// TIA Portal V20 export
DATA_BLOCK "HmiInterface"   // DB88
{ DB_Accessible_From_OPC_UA := 'FALSE' }
AUTHOR : ERsystem_FA2_DH. Kim
// stored: Access Published, DBAccessibleFromOPCUA false, DBAccessibleFromWebserver false, MemoryReserve 100, Namespace Unit1.Em7
   VAR
      em : "LAF_typeEmInterface";
      cm : Struct
         softCam : "Unit1.type_emRelations_em7_SoftCam";
         brakeTest : Struct
            sepaClampnCutterAxisZ : "LER_typeBrakeTestEmInterface";
            sepaGripperAxisZ : "LER_typeBrakeTestEmInterface";
            jrPusherAxisZ : "LER_typeBrakeTestEmInterface";
         END_STRUCT;
      END_STRUCT;
      sepaClamp : Struct
         jobs { S7_SetPoint := 'True'} : "LAF_typeJobsInterface";
         sequence { S7_SetPoint := 'True'} : "LAF_typeSequenceInterface";
      END_STRUCT;
      sepaGripper : Struct
         jobs { S7_SetPoint := 'True'} : "LAF_typeJobsInterface";
         sequence { S7_SetPoint := 'True'} : "LAF_typeSequenceInterface";
      END_STRUCT;
      jellyRollWinder : Struct
         jobs { S7_SetPoint := 'True'} : "LAF_typeJobsInterface";
         sequence { S7_SetPoint := 'True'} : "LAF_typeSequenceInterface";
      END_STRUCT;
      distance : Struct
         SepaClampToSepaGripperDisance : "LER_typeDistanceInterface";
         SepaGripperToSepaClampDisance : "LER_typeDistanceInterface";
         SepaGripperAxisCHomeDeg { S7_SetPoint := 'True'} : "LER_typeDistanceInterface";
         SepaGripperAxisXHomeDis { S7_SetPoint := 'True'} : "LER_typeDistanceInterface";
      END_STRUCT;
      cmSepaClampDetectSensor { S7_SetPoint := 'True'} : "LBC_typeDigitalSignalInterface";
      cmSepaGripperDetectSensor { S7_SetPoint := 'True'} : "LBC_typeDigitalSignalInterface";
      cmJRWinderDetectSensor { S7_SetPoint := 'True'} : "LBC_typeDigitalSignalInterface";
      cmSepaClampSafetyPinDetectSensor { S7_SetPoint := 'True'} : "LBC_typeDigitalSignalInterface";
      cmSepaGripperSafetyPinDetectSensor { S7_SetPoint := 'True'} : "LBC_typeDigitalSignalInterface";
   END_VAR
   VAR RETAIN
      cmSepaClampnCutterAxisX : "LBC_typeAxis64PosInterface";
      cmSepaClampnCutterAxisZ { S7_SetPoint := 'True'} : "LBC_typeAxis64PosInterface";
      cmSepaGripperAxisX : "LBC_typeAxis64PosInterface";
      cmSepaGripperAxisZ { S7_SetPoint := 'True'} : "LBC_typeAxis64PosInterface";
      cmSepaGripperAxisC : "LBC_typeAxis64PosInterface";
      cmJRWinderRearAxisY : "LBC_typeAxis64PosInterface";
      cmJRWinderFrontAxisY : "LBC_typeAxis64PosInterface";
      cmJRWinderAxisB { S7_SetPoint := 'True'} : "LBC_typeAxis64PosInterface";
      cmJRPusherAxisZ { S7_SetPoint := 'True'} : "LBC_typeAxis64PosInterface";
   END_VAR
   VAR
      cmSepaCutterUpDown { S7_SetPoint := 'True'} : "LBC_typeTwoWayActuatorInterface";
      cmSepaClampTopUpDown { S7_SetPoint := 'True'} : "LBC_typeTwoWayActuatorInterface";
      cmSepaClampBottomUpDown { S7_SetPoint := 'True'} : "LBC_typeTwoWayActuatorInterface";
      cmStackGripperOpenClose { S7_SetPoint := 'True'} : "LBC_typeTwoWayActuatorInterface";
      cmStackGripperFwdBwd { S7_SetPoint := 'True'} : "LBC_typeTwoWayActuatorInterface";
      cmJRWinderClampTopRearUpDown : "LBC_typeTwoWayActuatorInterface";
      cmJRWinderClampBtmRearUpDown : "LBC_typeTwoWayActuatorInterface";
      cmJRWinderClampTopFrontUpDown : "LBC_typeTwoWayActuatorInterface";
      cmJRWinderClampBtmFrontUpDown : "LBC_typeTwoWayActuatorInterface";
      cmPusherRollerUpDown : "LBC_typeTwoWayActuatorInterface";
      cmPusherRollerFwdBwd : "LBC_typeTwoWayActuatorInterface";
      cmHotWireCutter : "LER_typeHotWireCutterInterface";
      intCondition : Struct
         Axis_34 { S7_SetPoint := 'True'} : "LER.typeAxisIntlockAll";   // SepaClampnCutterAxisX
         Axis_35 { S7_SetPoint := 'True'} : "LER.typeAxisIntlockAll";   // SepaClampnCutterAxisZ
         Axis_36 { S7_SetPoint := 'True'} : "LER.typeAxisIntlockAll";   // SepaGripperAxisX
         Axis_37 { S7_SetPoint := 'True'} : "LER.typeAxisIntlockAll";   // SepaGripperAxisZ
         Axis_38 { S7_SetPoint := 'True'} : "LER.typeAxisIntlockAll";   // SepaGripperAxisC
         Axis_39 { S7_SetPoint := 'True'} : "LER.typeAxisIntlockAll";   // JRWinderFrontAxisY
         Axis_40 { S7_SetPoint := 'True'} : "LER.typeAxisIntlockAll";   // JRWinderRearAxisY
         Axis_41 { S7_SetPoint := 'True'} : "LER.typeAxisIntlockAll";   // JRWinderAxisB
         Axis_42 { S7_SetPoint := 'True'} : "LER.typeAxisIntlockAll";   // JRPusherAxisZ
         Axis_04 { S7_SetPoint := 'True'} : "LER.typeAxisIntlockAll";   // SepaClampnCutterAxisX
         Actuator_38 { S7_SetPoint := 'True'} : "LER.typeAxisActuatorCondition";   // SP
         Actuator_39 { S7_SetPoint := 'True'} : "LER.typeAxisActuatorCondition";   // SP
         Actuator_40 { S7_SetPoint := 'True'} : "LER.typeAxisActuatorCondition";   // JRWinderClampRightBtmUpDown
         Actuator_41 { S7_SetPoint := 'True'} : "LER.typeAxisActuatorCondition";   // JRWinderClampLeftBtmUpDown
         Actuator_42 { S7_SetPoint := 'True'} : "LER.typeAxisActuatorCondition";   // JRWinderClampLeftTopUpDown
         Actuator_43 { S7_SetPoint := 'True'} : "LER.typeAxisActuatorCondition";   // StackGripperFwdBwd
         Actuator_44 { S7_SetPoint := 'True'} : "LER.typeAxisActuatorCondition";   // SepaClampBottomUpDown
         Actuator_45 { S7_SetPoint := 'True'} : "LER.typeAxisActuatorCondition";   // SepaClampTopUpDown
         Actuator_46 { S7_SetPoint := 'True'} : "LER.typeAxisActuatorCondition";   // SepaCutterLeftUpDown
         Actuator_47 { S7_SetPoint := 'True'} : "LER.typeAxisActuatorCondition";   // JRWinderClampRightTopUpDown
         Actuator_48 { S7_SetPoint := 'True'} : "LER.typeAxisActuatorCondition";   // StackGripperOpenClose
         Actuator_49 { S7_SetPoint := 'True'} : "LER.typeAxisActuatorCondition";   // PusherRollerFwdBwd
      END_STRUCT;
   END_VAR
BEGIN
   em.interlinkMode.link := FALSE;
   em.interlinkMode.unlink := FALSE;
   em.interlinkMode.isLinked := TRUE;
   em.commands.enable := FALSE;
   em.commands.acknowledge := FALSE;
   em.commands.disableAlarms := FALSE;
   em.commands.activateSimulation := FALSE;
   em.commands.home := FALSE;
   em.commands.moveToInitialPosition := FALSE;
   em.commands.directModeControl := 16#0000_0001;
   em.commands.directStateControl := 16#0000_0004;
   em.status.enabled := TRUE;
   em.status.acknowledgeActive := FALSE;
   em.status.alarmsDisabled := FALSE;
   em.status.simulationActive := TRUE;
   em.status.safetyReleased := TRUE;
   em.status.initialized := FALSE;
   em.status.homed := FALSE;
   em.status.safeState := FALSE;
   em.status.stateComplete := FALSE;
   em.alarms.error := FALSE;
   em.alarms.warning := FALSE;
   em.alarms.info := FALSE;
   em.alarms.home := FALSE;
   cm.softCam.sepaClampnCutterAxisX.waitPos.inPos := TRUE;
   cm.softCam.sepaClampnCutterAxisX.waitPos.isBefore := FALSE;
   cm.softCam.sepaClampnCutterAxisX.waitPos.isAfter := FALSE;
   cm.softCam.sepaClampnCutterAxisX.sepaClampnCutPos.inPos := FALSE;
   cm.softCam.sepaClampnCutterAxisX.sepaClampnCutPos.isBefore := FALSE;
   cm.softCam.sepaClampnCutterAxisX.sepaClampnCutPos.isAfter := TRUE;
   cm.softCam.sepaClampnCutterAxisX.winderReadyPos.inPos := FALSE;
   cm.softCam.sepaClampnCutterAxisX.winderReadyPos.isBefore := TRUE;
   cm.softCam.sepaClampnCutterAxisX.winderReadyPos.isAfter := FALSE;
   cm.softCam.sepaClampnCutterAxisX.angle90.inPos := FALSE;
   cm.softCam.sepaClampnCutterAxisX.angle90.isBefore := TRUE;
   cm.softCam.sepaClampnCutterAxisX.angle90.isAfter := FALSE;
   cm.softCam.sepaClampnCutterAxisX.angle180.inPos := FALSE;
   cm.softCam.sepaClampnCutterAxisX.angle180.isBefore := TRUE;
   cm.softCam.sepaClampnCutterAxisX.angle180.isAfter := FALSE;
   cm.softCam.sepaClampnCutterAxisX.angle270.inPos := FALSE;
   cm.softCam.sepaClampnCutterAxisX.angle270.isBefore := TRUE;
   cm.softCam.sepaClampnCutterAxisX.angle270.isAfter := FALSE;
   cm.softCam.sepaClampnCutterAxisX.angle360.inPos := FALSE;
   cm.softCam.sepaClampnCutterAxisX.angle360.isBefore := TRUE;
   cm.softCam.sepaClampnCutterAxisX.angle360.isAfter := FALSE;
   cm.softCam.sepaClampnCutterAxisX.Pos8.inPos := FALSE;
   cm.softCam.sepaClampnCutterAxisX.Pos8.isBefore := FALSE;
   cm.softCam.sepaClampnCutterAxisX.Pos8.isAfter := TRUE;
   cm.softCam.sepaClampnCutterAxisX.Pos9.inPos := FALSE;
   cm.softCam.sepaClampnCutterAxisX.Pos9.isBefore := FALSE;
   cm.softCam.sepaClampnCutterAxisX.Pos9.isAfter := TRUE;
   cm.softCam.sepaClampnCutterAxisX.Pos10.inPos := FALSE;
   cm.softCam.sepaClampnCutterAxisX.Pos10.isBefore := FALSE;
   cm.softCam.sepaClampnCutterAxisX.Pos10.isAfter := TRUE;
   cm.softCam.sepaClampnCutterAxisX.Pos11.inPos := FALSE;
   cm.softCam.sepaClampnCutterAxisX.Pos11.isBefore := FALSE;
   cm.softCam.sepaClampnCutterAxisX.Pos11.isAfter := TRUE;
   cm.softCam.sepaClampnCutterAxisX.Pos12.inPos := FALSE;
   cm.softCam.sepaClampnCutterAxisX.Pos12.isBefore := FALSE;
   cm.softCam.sepaClampnCutterAxisX.Pos12.isAfter := TRUE;
   cm.softCam.sepaClampnCutterAxisX.Pos13.inPos := FALSE;
   cm.softCam.sepaClampnCutterAxisX.Pos13.isBefore := FALSE;
   cm.softCam.sepaClampnCutterAxisX.Pos13.isAfter := TRUE;
   cm.softCam.sepaClampnCutterAxisX.Pos14.inPos := FALSE;
   cm.softCam.sepaClampnCutterAxisX.Pos14.isBefore := FALSE;
   cm.softCam.sepaClampnCutterAxisX.Pos14.isAfter := TRUE;
   cm.softCam.sepaClampnCutterAxisX.Pos15.inPos := FALSE;
   cm.softCam.sepaClampnCutterAxisX.Pos15.isBefore := FALSE;
   cm.softCam.sepaClampnCutterAxisX.Pos15.isAfter := TRUE;
   cm.softCam.sepaClampnCutterAxisZ.waitPos.inPos := TRUE;
   cm.softCam.sepaClampnCutterAxisZ.waitPos.isBefore := FALSE;
   cm.softCam.sepaClampnCutterAxisZ.waitPos.isAfter := FALSE;
   cm.softCam.sepaClampnCutterAxisZ.sepaCutnClampPos.inPos := FALSE;
   cm.softCam.sepaClampnCutterAxisZ.sepaCutnClampPos.isBefore := TRUE;
   cm.softCam.sepaClampnCutterAxisZ.sepaCutnClampPos.isAfter := FALSE;
   cm.softCam.sepaClampnCutterAxisZ.winderReadyPos.inPos := FALSE;
   cm.softCam.sepaClampnCutterAxisZ.winderReadyPos.isBefore := TRUE;
   cm.softCam.sepaClampnCutterAxisZ.winderReadyPos.isAfter := FALSE;
   cm.softCam.sepaClampnCutterAxisZ.verticalPos.inPos := FALSE;
   cm.softCam.sepaClampnCutterAxisZ.verticalPos.isBefore := FALSE;
   cm.softCam.sepaClampnCutterAxisZ.verticalPos.isAfter := TRUE;
   cm.softCam.sepaClampnCutterAxisZ.horizonPos.inPos := TRUE;
   cm.softCam.sepaClampnCutterAxisZ.horizonPos.isBefore := FALSE;
   cm.softCam.sepaClampnCutterAxisZ.horizonPos.isAfter := FALSE;
   cm.softCam.sepaClampnCutterAxisZ.Pos5.inPos := TRUE;
   cm.softCam.sepaClampnCutterAxisZ.Pos5.isBefore := FALSE;
   cm.softCam.sepaClampnCutterAxisZ.Pos5.isAfter := FALSE;
   cm.softCam.sepaClampnCutterAxisZ.Pos6.inPos := TRUE;
   cm.softCam.sepaClampnCutterAxisZ.Pos6.isBefore := FALSE;
   cm.softCam.sepaClampnCutterAxisZ.Pos6.isAfter := FALSE;
   cm.softCam.sepaClampnCutterAxisZ.Pos7.inPos := TRUE;
   cm.softCam.sepaClampnCutterAxisZ.Pos7.isBefore := FALSE;
   cm.softCam.sepaClampnCutterAxisZ.Pos7.isAfter := FALSE;
   cm.softCam.sepaClampnCutterAxisZ.Pos8.inPos := TRUE;
   cm.softCam.sepaClampnCutterAxisZ.Pos8.isBefore := FALSE;
   cm.softCam.sepaClampnCutterAxisZ.Pos8.isAfter := FALSE;
   cm.softCam.sepaClampnCutterAxisZ.Pos9.inPos := TRUE;
   cm.softCam.sepaClampnCutterAxisZ.Pos9.isBefore := FALSE;
   cm.softCam.sepaClampnCutterAxisZ.Pos9.isAfter := FALSE;
   cm.softCam.sepaClampnCutterAxisZ.Pos10.inPos := TRUE;
   cm.softCam.sepaClampnCutterAxisZ.Pos10.isBefore := FALSE;
   cm.softCam.sepaClampnCutterAxisZ.Pos10.isAfter := FALSE;
   cm.softCam.sepaClampnCutterAxisZ.Pos11.inPos := TRUE;
   cm.softCam.sepaClampnCutterAxisZ.Pos11.isBefore := FALSE;
   cm.softCam.sepaClampnCutterAxisZ.Pos11.isAfter := FALSE;
   cm.softCam.sepaClampnCutterAxisZ.Pos12.inPos := TRUE;
   cm.softCam.sepaClampnCutterAxisZ.Pos12.isBefore := FALSE;
   cm.softCam.sepaClampnCutterAxisZ.Pos12.isAfter := FALSE;
   cm.softCam.sepaClampnCutterAxisZ.Pos13.inPos := TRUE;
   cm.softCam.sepaClampnCutterAxisZ.Pos13.isBefore := FALSE;
   cm.softCam.sepaClampnCutterAxisZ.Pos13.isAfter := FALSE;
   cm.softCam.sepaClampnCutterAxisZ.Pos14.inPos := TRUE;
   cm.softCam.sepaClampnCutterAxisZ.Pos14.isBefore := FALSE;
   cm.softCam.sepaClampnCutterAxisZ.Pos14.isAfter := FALSE;
   cm.softCam.sepaClampnCutterAxisZ.Pos15.inPos := TRUE;
   cm.softCam.sepaClampnCutterAxisZ.Pos15.isBefore := FALSE;
   cm.softCam.sepaClampnCutterAxisZ.Pos15.isAfter := FALSE;
   cm.softCam.sepaGripperAxisX.waitPos.inPos := TRUE;
   cm.softCam.sepaGripperAxisX.waitPos.isBefore := FALSE;
   cm.softCam.sepaGripperAxisX.waitPos.isAfter := FALSE;
   cm.softCam.sepaGripperAxisX.pickUpPOs.inPos := FALSE;
   cm.softCam.sepaGripperAxisX.pickUpPOs.isBefore := TRUE;
   cm.softCam.sepaGripperAxisX.pickUpPOs.isAfter := FALSE;
   cm.softCam.sepaGripperAxisX.sepaTailPos.inPos := FALSE;
   cm.softCam.sepaGripperAxisX.sepaTailPos.isBefore := TRUE;
   cm.softCam.sepaGripperAxisX.sepaTailPos.isAfter := FALSE;
   cm.softCam.sepaGripperAxisX.jrWinderPos.inPos := FALSE;
   cm.softCam.sepaGripperAxisX.jrWinderPos.isBefore := TRUE;
   cm.softCam.sepaGripperAxisX.jrWinderPos.isAfter := FALSE;
   cm.softCam.sepaGripperAxisX.turn_ngDischargePos.inPos := FALSE;
   cm.softCam.sepaGripperAxisX.turn_ngDischargePos.isBefore := TRUE;
   cm.softCam.sepaGripperAxisX.turn_ngDischargePos.isAfter := FALSE;
   cm.softCam.sepaGripperAxisX.avoidPos.inPos := TRUE;
   cm.softCam.sepaGripperAxisX.avoidPos.isBefore := FALSE;
   cm.softCam.sepaGripperAxisX.avoidPos.isAfter := FALSE;
   cm.softCam.sepaGripperAxisX.okDisChargePos.inPos := FALSE;
   cm.softCam.sepaGripperAxisX.okDisChargePos.isBefore := FALSE;
   cm.softCam.sepaGripperAxisX.okDisChargePos.isAfter := TRUE;
   cm.softCam.sepaGripperAxisX.ngSepaTailPos.inPos := FALSE;
   cm.softCam.sepaGripperAxisX.ngSepaTailPos.isBefore := FALSE;
   cm.softCam.sepaGripperAxisX.ngSepaTailPos.isAfter := TRUE;
   cm.softCam.sepaGripperAxisX.jrWinderZonePos.inPos := FALSE;
   cm.softCam.sepaGripperAxisX.jrWinderZonePos.isBefore := FALSE;
   cm.softCam.sepaGripperAxisX.jrWinderZonePos.isAfter := TRUE;
   cm.softCam.sepaGripperAxisX.gripperAxisCCollisionZonePos.inPos := FALSE;
   cm.softCam.sepaGripperAxisX.gripperAxisCCollisionZonePos.isBefore := FALSE;
   cm.softCam.sepaGripperAxisX.gripperAxisCCollisionZonePos.isAfter := TRUE;
   cm.softCam.sepaGripperAxisX.anodePnPZonePos.inPos := FALSE;
   cm.softCam.sepaGripperAxisX.anodePnPZonePos.isBefore := FALSE;
   cm.softCam.sepaGripperAxisX.anodePnPZonePos.isAfter := TRUE;
   cm.softCam.sepaGripperAxisX.pickUpBeforePos.inPos := FALSE;
   cm.softCam.sepaGripperAxisX.pickUpBeforePos.isBefore := FALSE;
   cm.softCam.sepaGripperAxisX.pickUpBeforePos.isAfter := TRUE;
   cm.softCam.sepaGripperAxisX.Pos12.inPos := FALSE;
   cm.softCam.sepaGripperAxisX.Pos12.isBefore := FALSE;
   cm.softCam.sepaGripperAxisX.Pos12.isAfter := TRUE;
   cm.softCam.sepaGripperAxisX.Pos13.inPos := FALSE;
   cm.softCam.sepaGripperAxisX.Pos13.isBefore := FALSE;
   cm.softCam.sepaGripperAxisX.Pos13.isAfter := TRUE;
   cm.softCam.sepaGripperAxisX.Pos14.inPos := FALSE;
   cm.softCam.sepaGripperAxisX.Pos14.isBefore := FALSE;
   cm.softCam.sepaGripperAxisX.Pos14.isAfter := TRUE;
   cm.softCam.sepaGripperAxisX.Pos15.inPos := FALSE;
   cm.softCam.sepaGripperAxisX.Pos15.isBefore := FALSE;
   cm.softCam.sepaGripperAxisX.Pos15.isAfter := TRUE;
   cm.softCam.sepaGripperAxisZ.waitPos.inPos := TRUE;
   cm.softCam.sepaGripperAxisZ.waitPos.isBefore := FALSE;
   cm.softCam.sepaGripperAxisZ.waitPos.isAfter := FALSE;
   cm.softCam.sepaGripperAxisZ.jrWinderPos.inPos := FALSE;
   cm.softCam.sepaGripperAxisZ.jrWinderPos.isBefore := TRUE;
   cm.softCam.sepaGripperAxisZ.jrWinderPos.isAfter := FALSE;
   cm.softCam.sepaGripperAxisZ.turnPos.inPos := FALSE;
   cm.softCam.sepaGripperAxisZ.turnPos.isBefore := TRUE;
   cm.softCam.sepaGripperAxisZ.turnPos.isAfter := FALSE;
   cm.softCam.sepaGripperAxisZ.jrWinderRePickUpPos.inPos := FALSE;
   cm.softCam.sepaGripperAxisZ.jrWinderRePickUpPos.isBefore := TRUE;
   cm.softCam.sepaGripperAxisZ.jrWinderRePickUpPos.isAfter := FALSE;
   cm.softCam.sepaGripperAxisZ.okDisChargePos.inPos := FALSE;
   cm.softCam.sepaGripperAxisZ.okDisChargePos.isBefore := TRUE;
   cm.softCam.sepaGripperAxisZ.okDisChargePos.isAfter := FALSE;
   cm.softCam.sepaGripperAxisZ.ngDischargePos.inPos := FALSE;
   cm.softCam.sepaGripperAxisZ.ngDischargePos.isBefore := TRUE;
   cm.softCam.sepaGripperAxisZ.ngDischargePos.isAfter := FALSE;
   cm.softCam.sepaGripperAxisZ.pickUpPos.inPos := FALSE;
   cm.softCam.sepaGripperAxisZ.pickUpPos.isBefore := TRUE;
   cm.softCam.sepaGripperAxisZ.pickUpPos.isAfter := FALSE;
   cm.softCam.sepaGripperAxisZ.Pos7.inPos := TRUE;
   cm.softCam.sepaGripperAxisZ.Pos7.isBefore := FALSE;
   cm.softCam.sepaGripperAxisZ.Pos7.isAfter := FALSE;
   cm.softCam.sepaGripperAxisZ.Pos8.inPos := TRUE;
   cm.softCam.sepaGripperAxisZ.Pos8.isBefore := FALSE;
   cm.softCam.sepaGripperAxisZ.Pos8.isAfter := FALSE;
   cm.softCam.sepaGripperAxisZ.Pos9.inPos := TRUE;
   cm.softCam.sepaGripperAxisZ.Pos9.isBefore := FALSE;
   cm.softCam.sepaGripperAxisZ.Pos9.isAfter := FALSE;
   cm.softCam.sepaGripperAxisZ.Pos10.inPos := TRUE;
   cm.softCam.sepaGripperAxisZ.Pos10.isBefore := FALSE;
   cm.softCam.sepaGripperAxisZ.Pos10.isAfter := FALSE;
   cm.softCam.sepaGripperAxisZ.Pos11.inPos := TRUE;
   cm.softCam.sepaGripperAxisZ.Pos11.isBefore := FALSE;
   cm.softCam.sepaGripperAxisZ.Pos11.isAfter := FALSE;
   cm.softCam.sepaGripperAxisZ.Pos12.inPos := TRUE;
   cm.softCam.sepaGripperAxisZ.Pos12.isBefore := FALSE;
   cm.softCam.sepaGripperAxisZ.Pos12.isAfter := FALSE;
   cm.softCam.sepaGripperAxisZ.Pos13.inPos := TRUE;
   cm.softCam.sepaGripperAxisZ.Pos13.isBefore := FALSE;
   cm.softCam.sepaGripperAxisZ.Pos13.isAfter := FALSE;
   cm.softCam.sepaGripperAxisZ.Pos14.inPos := TRUE;
   cm.softCam.sepaGripperAxisZ.Pos14.isBefore := FALSE;
   cm.softCam.sepaGripperAxisZ.Pos14.isAfter := FALSE;
   cm.softCam.sepaGripperAxisZ.Pos15.inPos := TRUE;
   cm.softCam.sepaGripperAxisZ.Pos15.isBefore := FALSE;
   cm.softCam.sepaGripperAxisZ.Pos15.isAfter := FALSE;
   cm.softCam.sepaGripperAxisC.waitPos.inPos := TRUE;
   cm.softCam.sepaGripperAxisC.waitPos.isBefore := FALSE;
   cm.softCam.sepaGripperAxisC.waitPos.isAfter := FALSE;
   cm.softCam.sepaGripperAxisC.okDischargePos.inPos := FALSE;
   cm.softCam.sepaGripperAxisC.okDischargePos.isBefore := TRUE;
   cm.softCam.sepaGripperAxisC.okDischargePos.isAfter := FALSE;
   cm.softCam.sepaGripperAxisC.ngDischargePos.inPos := FALSE;
   cm.softCam.sepaGripperAxisC.ngDischargePos.isBefore := TRUE;
   cm.softCam.sepaGripperAxisC.ngDischargePos.isAfter := FALSE;
   cm.softCam.sepaGripperAxisC.Pos3.inPos := TRUE;
   cm.softCam.sepaGripperAxisC.Pos3.isBefore := FALSE;
   cm.softCam.sepaGripperAxisC.Pos3.isAfter := FALSE;
   cm.softCam.sepaGripperAxisC.Pos4.inPos := TRUE;
   cm.softCam.sepaGripperAxisC.Pos4.isBefore := FALSE;
   cm.softCam.sepaGripperAxisC.Pos4.isAfter := FALSE;
   cm.softCam.sepaGripperAxisC.Pos5.inPos := TRUE;
   cm.softCam.sepaGripperAxisC.Pos5.isBefore := FALSE;
   cm.softCam.sepaGripperAxisC.Pos5.isAfter := FALSE;
   cm.softCam.sepaGripperAxisC.Pos6.inPos := TRUE;
   cm.softCam.sepaGripperAxisC.Pos6.isBefore := FALSE;
   cm.softCam.sepaGripperAxisC.Pos6.isAfter := FALSE;
   cm.softCam.sepaGripperAxisC.Pos7.inPos := TRUE;
   cm.softCam.sepaGripperAxisC.Pos7.isBefore := FALSE;
   cm.softCam.sepaGripperAxisC.Pos7.isAfter := FALSE;
   cm.softCam.sepaGripperAxisC.Pos8.inPos := TRUE;
   cm.softCam.sepaGripperAxisC.Pos8.isBefore := FALSE;
   cm.softCam.sepaGripperAxisC.Pos8.isAfter := FALSE;
   cm.softCam.sepaGripperAxisC.Pos9.inPos := TRUE;
   cm.softCam.sepaGripperAxisC.Pos9.isBefore := FALSE;
   cm.softCam.sepaGripperAxisC.Pos9.isAfter := FALSE;
   cm.softCam.sepaGripperAxisC.Pos10.inPos := TRUE;
   cm.softCam.sepaGripperAxisC.Pos10.isBefore := FALSE;
   cm.softCam.sepaGripperAxisC.Pos10.isAfter := FALSE;
   cm.softCam.sepaGripperAxisC.Pos11.inPos := TRUE;
   cm.softCam.sepaGripperAxisC.Pos11.isBefore := FALSE;
   cm.softCam.sepaGripperAxisC.Pos11.isAfter := FALSE;
   cm.softCam.sepaGripperAxisC.Pos12.inPos := TRUE;
   cm.softCam.sepaGripperAxisC.Pos12.isBefore := FALSE;
   cm.softCam.sepaGripperAxisC.Pos12.isAfter := FALSE;
   cm.softCam.sepaGripperAxisC.Pos13.inPos := TRUE;
   cm.softCam.sepaGripperAxisC.Pos13.isBefore := FALSE;
   cm.softCam.sepaGripperAxisC.Pos13.isAfter := FALSE;
   cm.softCam.sepaGripperAxisC.Pos14.inPos := TRUE;
   cm.softCam.sepaGripperAxisC.Pos14.isBefore := FALSE;
   cm.softCam.sepaGripperAxisC.Pos14.isAfter := FALSE;
   cm.softCam.sepaGripperAxisC.Pos15.inPos := TRUE;
   cm.softCam.sepaGripperAxisC.Pos15.isBefore := FALSE;
   cm.softCam.sepaGripperAxisC.Pos15.isAfter := FALSE;
   cm.softCam.jrWinderRearAxisY.waitPos.inPos := TRUE;
   cm.softCam.jrWinderRearAxisY.waitPos.isBefore := FALSE;
   cm.softCam.jrWinderRearAxisY.waitPos.isAfter := FALSE;
   cm.softCam.jrWinderRearAxisY.clampPos.inPos := FALSE;
   cm.softCam.jrWinderRearAxisY.clampPos.isBefore := TRUE;
   cm.softCam.jrWinderRearAxisY.clampPos.isAfter := FALSE;
   cm.softCam.jrWinderRearAxisY.Pos2.inPos := TRUE;
   cm.softCam.jrWinderRearAxisY.Pos2.isBefore := FALSE;
   cm.softCam.jrWinderRearAxisY.Pos2.isAfter := FALSE;
   cm.softCam.jrWinderRearAxisY.Pos3.inPos := TRUE;
   cm.softCam.jrWinderRearAxisY.Pos3.isBefore := FALSE;
   cm.softCam.jrWinderRearAxisY.Pos3.isAfter := FALSE;
   cm.softCam.jrWinderRearAxisY.Pos4.inPos := TRUE;
   cm.softCam.jrWinderRearAxisY.Pos4.isBefore := FALSE;
   cm.softCam.jrWinderRearAxisY.Pos4.isAfter := FALSE;
   cm.softCam.jrWinderRearAxisY.Pos5.inPos := TRUE;
   cm.softCam.jrWinderRearAxisY.Pos5.isBefore := FALSE;
   cm.softCam.jrWinderRearAxisY.Pos5.isAfter := FALSE;
   cm.softCam.jrWinderRearAxisY.Pos6.inPos := TRUE;
   cm.softCam.jrWinderRearAxisY.Pos6.isBefore := FALSE;
   cm.softCam.jrWinderRearAxisY.Pos6.isAfter := FALSE;
   cm.softCam.jrWinderRearAxisY.Pos7.inPos := TRUE;
   cm.softCam.jrWinderRearAxisY.Pos7.isBefore := FALSE;
   cm.softCam.jrWinderRearAxisY.Pos7.isAfter := FALSE;
   cm.softCam.jrWinderRearAxisY.Pos8.inPos := TRUE;
   cm.softCam.jrWinderRearAxisY.Pos8.isBefore := FALSE;
   cm.softCam.jrWinderRearAxisY.Pos8.isAfter := FALSE;
   cm.softCam.jrWinderRearAxisY.Pos9.inPos := TRUE;
   cm.softCam.jrWinderRearAxisY.Pos9.isBefore := FALSE;
   cm.softCam.jrWinderRearAxisY.Pos9.isAfter := FALSE;
   cm.softCam.jrWinderRearAxisY.Pos10.inPos := TRUE;
   cm.softCam.jrWinderRearAxisY.Pos10.isBefore := FALSE;
   cm.softCam.jrWinderRearAxisY.Pos10.isAfter := FALSE;
   cm.softCam.jrWinderRearAxisY.Pos11.inPos := TRUE;
   cm.softCam.jrWinderRearAxisY.Pos11.isBefore := FALSE;
   cm.softCam.jrWinderRearAxisY.Pos11.isAfter := FALSE;
   cm.softCam.jrWinderRearAxisY.Pos12.inPos := TRUE;
   cm.softCam.jrWinderRearAxisY.Pos12.isBefore := FALSE;
   cm.softCam.jrWinderRearAxisY.Pos12.isAfter := FALSE;
   cm.softCam.jrWinderRearAxisY.Pos13.inPos := TRUE;
   cm.softCam.jrWinderRearAxisY.Pos13.isBefore := FALSE;
   cm.softCam.jrWinderRearAxisY.Pos13.isAfter := FALSE;
   cm.softCam.jrWinderRearAxisY.Pos14.inPos := TRUE;
   cm.softCam.jrWinderRearAxisY.Pos14.isBefore := FALSE;
   cm.softCam.jrWinderRearAxisY.Pos14.isAfter := FALSE;
   cm.softCam.jrWinderRearAxisY.Pos15.inPos := TRUE;
   cm.softCam.jrWinderRearAxisY.Pos15.isBefore := FALSE;
   cm.softCam.jrWinderRearAxisY.Pos15.isAfter := FALSE;
   cm.softCam.jrWinderFrontAxisY.waitPos.inPos := TRUE;
   cm.softCam.jrWinderFrontAxisY.waitPos.isBefore := FALSE;
   cm.softCam.jrWinderFrontAxisY.waitPos.isAfter := FALSE;
   cm.softCam.jrWinderFrontAxisY.clampPos.inPos := FALSE;
   cm.softCam.jrWinderFrontAxisY.clampPos.isBefore := TRUE;
   cm.softCam.jrWinderFrontAxisY.clampPos.isAfter := FALSE;
   cm.softCam.jrWinderFrontAxisY.Pos2.inPos := TRUE;
   cm.softCam.jrWinderFrontAxisY.Pos2.isBefore := FALSE;
   cm.softCam.jrWinderFrontAxisY.Pos2.isAfter := FALSE;
   cm.softCam.jrWinderFrontAxisY.Pos3.inPos := TRUE;
   cm.softCam.jrWinderFrontAxisY.Pos3.isBefore := FALSE;
   cm.softCam.jrWinderFrontAxisY.Pos3.isAfter := FALSE;
   cm.softCam.jrWinderFrontAxisY.Pos4.inPos := TRUE;
   cm.softCam.jrWinderFrontAxisY.Pos4.isBefore := FALSE;
   cm.softCam.jrWinderFrontAxisY.Pos4.isAfter := FALSE;
   cm.softCam.jrWinderFrontAxisY.Pos5.inPos := TRUE;
   cm.softCam.jrWinderFrontAxisY.Pos5.isBefore := FALSE;
   cm.softCam.jrWinderFrontAxisY.Pos5.isAfter := FALSE;
   cm.softCam.jrWinderFrontAxisY.Pos6.inPos := TRUE;
   cm.softCam.jrWinderFrontAxisY.Pos6.isBefore := FALSE;
   cm.softCam.jrWinderFrontAxisY.Pos6.isAfter := FALSE;
   cm.softCam.jrWinderFrontAxisY.Pos7.inPos := TRUE;
   cm.softCam.jrWinderFrontAxisY.Pos7.isBefore := FALSE;
   cm.softCam.jrWinderFrontAxisY.Pos7.isAfter := FALSE;
   cm.softCam.jrWinderFrontAxisY.Pos8.inPos := TRUE;
   cm.softCam.jrWinderFrontAxisY.Pos8.isBefore := FALSE;
   cm.softCam.jrWinderFrontAxisY.Pos8.isAfter := FALSE;
   cm.softCam.jrWinderFrontAxisY.Pos9.inPos := TRUE;
   cm.softCam.jrWinderFrontAxisY.Pos9.isBefore := FALSE;
   cm.softCam.jrWinderFrontAxisY.Pos9.isAfter := FALSE;
   cm.softCam.jrWinderFrontAxisY.Pos10.inPos := TRUE;
   cm.softCam.jrWinderFrontAxisY.Pos10.isBefore := FALSE;
   cm.softCam.jrWinderFrontAxisY.Pos10.isAfter := FALSE;
   cm.softCam.jrWinderFrontAxisY.Pos11.inPos := TRUE;
   cm.softCam.jrWinderFrontAxisY.Pos11.isBefore := FALSE;
   cm.softCam.jrWinderFrontAxisY.Pos11.isAfter := FALSE;
   cm.softCam.jrWinderFrontAxisY.Pos12.inPos := TRUE;
   cm.softCam.jrWinderFrontAxisY.Pos12.isBefore := FALSE;
   cm.softCam.jrWinderFrontAxisY.Pos12.isAfter := FALSE;
   cm.softCam.jrWinderFrontAxisY.Pos13.inPos := TRUE;
   cm.softCam.jrWinderFrontAxisY.Pos13.isBefore := FALSE;
   cm.softCam.jrWinderFrontAxisY.Pos13.isAfter := FALSE;
   cm.softCam.jrWinderFrontAxisY.Pos14.inPos := TRUE;
   cm.softCam.jrWinderFrontAxisY.Pos14.isBefore := FALSE;
   cm.softCam.jrWinderFrontAxisY.Pos14.isAfter := FALSE;
   cm.softCam.jrWinderFrontAxisY.Pos15.inPos := TRUE;
   cm.softCam.jrWinderFrontAxisY.Pos15.isBefore := FALSE;
   cm.softCam.jrWinderFrontAxisY.Pos15.isAfter := FALSE;
   cm.softCam.jrWinderAxisB.waitPos.inPos := TRUE;
   cm.softCam.jrWinderAxisB.waitPos.isBefore := FALSE;
   cm.softCam.jrWinderAxisB.waitPos.isAfter := FALSE;
   cm.softCam.jrWinderAxisB.angle90.inPos := FALSE;
   cm.softCam.jrWinderAxisB.angle90.isBefore := TRUE;
   cm.softCam.jrWinderAxisB.angle90.isAfter := FALSE;
   cm.softCam.jrWinderAxisB.angle180.inPos := FALSE;
   cm.softCam.jrWinderAxisB.angle180.isBefore := TRUE;
   cm.softCam.jrWinderAxisB.angle180.isAfter := FALSE;
   cm.softCam.jrWinderAxisB.angle270.inPos := FALSE;
   cm.softCam.jrWinderAxisB.angle270.isBefore := TRUE;
   cm.softCam.jrWinderAxisB.angle270.isAfter := FALSE;
   cm.softCam.jrWinderAxisB.angle360.inPos := TRUE;
   cm.softCam.jrWinderAxisB.angle360.isBefore := FALSE;
   cm.softCam.jrWinderAxisB.angle360.isAfter := FALSE;
   cm.softCam.jrWinderAxisB.angle450.inPos := TRUE;
   cm.softCam.jrWinderAxisB.angle450.isBefore := FALSE;
   cm.softCam.jrWinderAxisB.angle450.isAfter := FALSE;
   cm.softCam.jrWinderAxisB.angle540.inPos := TRUE;
   cm.softCam.jrWinderAxisB.angle540.isBefore := FALSE;
   cm.softCam.jrWinderAxisB.angle540.isAfter := FALSE;
   cm.softCam.jrWinderAxisB.Pos9.inPos := TRUE;
   cm.softCam.jrWinderAxisB.Pos9.isBefore := FALSE;
   cm.softCam.jrWinderAxisB.Pos9.isAfter := FALSE;
   cm.softCam.jrWinderAxisB.Pos10.inPos := TRUE;
   cm.softCam.jrWinderAxisB.Pos10.isBefore := FALSE;
   cm.softCam.jrWinderAxisB.Pos10.isAfter := FALSE;
   cm.softCam.jrWinderAxisB.Pos11.inPos := TRUE;
   cm.softCam.jrWinderAxisB.Pos11.isBefore := FALSE;
   cm.softCam.jrWinderAxisB.Pos11.isAfter := FALSE;
   cm.softCam.jrWinderAxisB.Pos12.inPos := TRUE;
   cm.softCam.jrWinderAxisB.Pos12.isBefore := FALSE;
   cm.softCam.jrWinderAxisB.Pos12.isAfter := FALSE;
   cm.softCam.jrWinderAxisB.Pos13.inPos := TRUE;
   cm.softCam.jrWinderAxisB.Pos13.isBefore := FALSE;
   cm.softCam.jrWinderAxisB.Pos13.isAfter := FALSE;
   cm.softCam.jrWinderAxisB.Pos14.inPos := TRUE;
   cm.softCam.jrWinderAxisB.Pos14.isBefore := FALSE;
   cm.softCam.jrWinderAxisB.Pos14.isAfter := FALSE;
   cm.softCam.jrWinderAxisB.Pos15.inPos := TRUE;
   cm.softCam.jrWinderAxisB.Pos15.isBefore := FALSE;
   cm.softCam.jrWinderAxisB.Pos15.isAfter := FALSE;
   cm.softCam.jrPusherAxisZ.waitPos.inPos := TRUE;
   cm.softCam.jrPusherAxisZ.waitPos.isBefore := FALSE;
   cm.softCam.jrPusherAxisZ.waitPos.isAfter := FALSE;
   cm.softCam.jrPusherAxisZ.downPos.inPos := FALSE;
   cm.softCam.jrPusherAxisZ.downPos.isBefore := TRUE;
   cm.softCam.jrPusherAxisZ.downPos.isAfter := FALSE;
   cm.softCam.jrPusherAxisZ.verticalPos.inPos := FALSE;
   cm.softCam.jrPusherAxisZ.verticalPos.isBefore := FALSE;
   cm.softCam.jrPusherAxisZ.verticalPos.isAfter := TRUE;
   cm.softCam.jrPusherAxisZ.horizonPos.inPos := TRUE;
   cm.softCam.jrPusherAxisZ.horizonPos.isBefore := FALSE;
   cm.softCam.jrPusherAxisZ.horizonPos.isAfter := FALSE;
   cm.softCam.jrPusherAxisZ.Pos4.inPos := TRUE;
   cm.softCam.jrPusherAxisZ.Pos4.isBefore := FALSE;
   cm.softCam.jrPusherAxisZ.Pos4.isAfter := FALSE;
   cm.softCam.jrPusherAxisZ.Pos5.inPos := TRUE;
   cm.softCam.jrPusherAxisZ.Pos5.isBefore := FALSE;
   cm.softCam.jrPusherAxisZ.Pos5.isAfter := FALSE;
   cm.softCam.jrPusherAxisZ.Pos6.inPos := TRUE;
   cm.softCam.jrPusherAxisZ.Pos6.isBefore := FALSE;
   cm.softCam.jrPusherAxisZ.Pos6.isAfter := FALSE;
   cm.softCam.jrPusherAxisZ.Pos7.inPos := TRUE;
   cm.softCam.jrPusherAxisZ.Pos7.isBefore := FALSE;
   cm.softCam.jrPusherAxisZ.Pos7.isAfter := FALSE;
   cm.softCam.jrPusherAxisZ.Pos8.inPos := TRUE;
   cm.softCam.jrPusherAxisZ.Pos8.isBefore := FALSE;
   cm.softCam.jrPusherAxisZ.Pos8.isAfter := FALSE;
   cm.softCam.jrPusherAxisZ.Pos9.inPos := TRUE;
   cm.softCam.jrPusherAxisZ.Pos9.isBefore := FALSE;
   cm.softCam.jrPusherAxisZ.Pos9.isAfter := FALSE;
   cm.softCam.jrPusherAxisZ.Pos10.inPos := TRUE;
   cm.softCam.jrPusherAxisZ.Pos10.isBefore := FALSE;
   cm.softCam.jrPusherAxisZ.Pos10.isAfter := FALSE;
   cm.softCam.jrPusherAxisZ.Pos11.inPos := TRUE;
   cm.softCam.jrPusherAxisZ.Pos11.isBefore := FALSE;
   cm.softCam.jrPusherAxisZ.Pos11.isAfter := FALSE;
   cm.softCam.jrPusherAxisZ.Pos12.inPos := TRUE;
   cm.softCam.jrPusherAxisZ.Pos12.isBefore := FALSE;
   cm.softCam.jrPusherAxisZ.Pos12.isAfter := FALSE;
   cm.softCam.jrPusherAxisZ.Pos13.inPos := TRUE;
   cm.softCam.jrPusherAxisZ.Pos13.isBefore := FALSE;
   cm.softCam.jrPusherAxisZ.Pos13.isAfter := FALSE;
   cm.softCam.jrPusherAxisZ.Pos14.inPos := TRUE;
   cm.softCam.jrPusherAxisZ.Pos14.isBefore := FALSE;
   cm.softCam.jrPusherAxisZ.Pos14.isAfter := FALSE;
   cm.softCam.jrPusherAxisZ.Pos15.inPos := TRUE;
   cm.softCam.jrPusherAxisZ.Pos15.isBefore := FALSE;
   cm.softCam.jrPusherAxisZ.Pos15.isAfter := FALSE;
   cm.brakeTest.sepaClampnCutterAxisZ.commands.start := FALSE;
   cm.brakeTest.sepaClampnCutterAxisZ.commands.stop := FALSE;
   cm.brakeTest.sepaClampnCutterAxisZ.monitoring.error := FALSE;
   cm.brakeTest.sepaClampnCutterAxisZ.monitoring.ready := FALSE;
   cm.brakeTest.sepaClampnCutterAxisZ.monitoring.busy := FALSE;
   cm.brakeTest.sepaClampnCutterAxisZ.monitoring.complete := FALSE;
   cm.brakeTest.sepaClampnCutterAxisZ.monitoring.brakeSelected := FALSE;
   cm.brakeTest.sepaClampnCutterAxisZ.monitoring.brakeActive := FALSE;
   cm.brakeTest.sepaClampnCutterAxisZ.monitoring.brakeResult := FALSE;
   cm.brakeTest.sepaClampnCutterAxisZ.monitoring.brakeCompleted := FALSE;
   cm.brakeTest.sepaClampnCutterAxisZ.monitoring."step" := 0;
   cm.brakeTest.sepaGripperAxisZ.commands.start := FALSE;
   cm.brakeTest.sepaGripperAxisZ.commands.stop := FALSE;
   cm.brakeTest.sepaGripperAxisZ.monitoring.error := FALSE;
   cm.brakeTest.sepaGripperAxisZ.monitoring.ready := FALSE;
   cm.brakeTest.sepaGripperAxisZ.monitoring.busy := FALSE;
   cm.brakeTest.sepaGripperAxisZ.monitoring.complete := FALSE;
   cm.brakeTest.sepaGripperAxisZ.monitoring.brakeSelected := FALSE;
   cm.brakeTest.sepaGripperAxisZ.monitoring.brakeActive := FALSE;
   cm.brakeTest.sepaGripperAxisZ.monitoring.brakeResult := FALSE;
   cm.brakeTest.sepaGripperAxisZ.monitoring.brakeCompleted := FALSE;
   cm.brakeTest.sepaGripperAxisZ.monitoring."step" := 0;
   cm.brakeTest.jrPusherAxisZ.commands.start := FALSE;
   cm.brakeTest.jrPusherAxisZ.commands.stop := FALSE;
   cm.brakeTest.jrPusherAxisZ.monitoring.error := FALSE;
   cm.brakeTest.jrPusherAxisZ.monitoring.ready := FALSE;
   cm.brakeTest.jrPusherAxisZ.monitoring.busy := FALSE;
   cm.brakeTest.jrPusherAxisZ.monitoring.complete := FALSE;
   cm.brakeTest.jrPusherAxisZ.monitoring.brakeSelected := FALSE;
   cm.brakeTest.jrPusherAxisZ.monitoring.brakeActive := FALSE;
   cm.brakeTest.jrPusherAxisZ.monitoring.brakeResult := FALSE;
   cm.brakeTest.jrPusherAxisZ.monitoring.brakeCompleted := FALSE;
   cm.brakeTest.jrPusherAxisZ.monitoring."step" := 0;
   sepaClamp.jobs.commands.setJobNumber := 0;
   sepaClamp.jobs.commands.reset := FALSE;
   sepaClamp.jobs.status.activeJobNumber := 1;
   sepaClamp.jobs.status.previousCycleJobNumber := 1;
   sepaClamp.jobs.status.manualControlEnabled := FALSE;
   sepaClamp.jobs.status.memoryJobTime := 16#0000_4E90_6672_4E37;
   sepaClamp.sequence.commands.setAutomaticMode := FALSE;
   sepaClamp.sequence.commands.setSingleStepMode := FALSE;
   sepaClamp.sequence.commands.off := FALSE;
   sepaClamp.sequence.commands.initialize := FALSE;
   sepaClamp.sequence.commands.start := FALSE;
   sepaClamp.sequence.commands.immediateStop := FALSE;
   sepaClamp.sequence.commands.hold := FALSE;
   sepaClamp.sequence.commands.nextStep := FALSE;
   sepaClamp.sequence.commands.interlockStepChange := FALSE;
   sepaClamp.sequence.monitoring.automaticMode := TRUE;
   sepaClamp.sequence.monitoring.singleStepMode := FALSE;
   sepaClamp.sequence.monitoring.currentStep := 101;
   sepaClamp.sequence.monitoring.nextStep := 101;
   sepaClamp.sequence.monitoring.previousStep := 1;
   sepaClamp.sequence.monitoring.currentStepSTRING := 'N/A';
   sepaClamp.sequence.monitoring.nextStepSTRING := 'N/A';
   sepaClamp.sequence.monitoring.previousStepSTRING := 'N/A';
   sepaClamp.sequence.monitoring.inStepIdle := FALSE;
   sepaClamp.sequence.monitoring.inStepStopped := FALSE;
   sepaClamp.sequence.monitoring.seqActive := TRUE;
   sepaClamp.sequence.monitoring.stepActive := TRUE;
   sepaClamp.sequence.monitoring.stepComplete := FALSE;
   sepaClamp.sequence.monitoring.executionEnabled := FALSE;
   sepaClamp.sequence.monitoring.initRequired := FALSE;
   sepaClamp.sequence.monitoring.stepChangeReleased := TRUE;
   sepaClamp.sequence.monitoring.justSteppedPulse := FALSE;
   sepaClamp.sequence.monitoring.manualControlEnabled := FALSE;
   sepaClamp.sequence.monitoring.manualModeChangeEnabled := FALSE;
   sepaClamp.sequence.monitoring.memoryStepTimer := 16#0000_4E90_6828_A4A1;
   sepaGripper.jobs.commands.setJobNumber := 0;
   sepaGripper.jobs.commands.reset := FALSE;
   sepaGripper.jobs.status.activeJobNumber := 0;
   sepaGripper.jobs.status.previousCycleJobNumber := 0;
   sepaGripper.jobs.status.manualControlEnabled := FALSE;
   sepaGripper.jobs.status.memoryJobTime := 16#0000_4E92_AEA1_93D2;
   sepaGripper.sequence.commands.setAutomaticMode := FALSE;
   sepaGripper.sequence.commands.setSingleStepMode := FALSE;
   sepaGripper.sequence.commands.off := FALSE;
   sepaGripper.sequence.commands.initialize := FALSE;
   sepaGripper.sequence.commands.start := FALSE;
   sepaGripper.sequence.commands.immediateStop := FALSE;
   sepaGripper.sequence.commands.hold := FALSE;
   sepaGripper.sequence.commands.nextStep := FALSE;
   sepaGripper.sequence.commands.interlockStepChange := FALSE;
   sepaGripper.sequence.monitoring.automaticMode := TRUE;
   sepaGripper.sequence.monitoring.singleStepMode := FALSE;
   sepaGripper.sequence.monitoring.currentStep := 1;
   sepaGripper.sequence.monitoring.nextStep := 1;
   sepaGripper.sequence.monitoring.previousStep := 190;
   sepaGripper.sequence.monitoring.currentStepSTRING := 'N/A';
   sepaGripper.sequence.monitoring.nextStepSTRING := 'N/A';
   sepaGripper.sequence.monitoring.previousStepSTRING := 'N/A';
   sepaGripper.sequence.monitoring.inStepIdle := TRUE;
   sepaGripper.sequence.monitoring.inStepStopped := FALSE;
   sepaGripper.sequence.monitoring.seqActive := TRUE;
   sepaGripper.sequence.monitoring.stepActive := TRUE;
   sepaGripper.sequence.monitoring.stepComplete := FALSE;
   sepaGripper.sequence.monitoring.executionEnabled := TRUE;
   sepaGripper.sequence.monitoring.initRequired := FALSE;
   sepaGripper.sequence.monitoring.stepChangeReleased := TRUE;
   sepaGripper.sequence.monitoring.justSteppedPulse := FALSE;
   sepaGripper.sequence.monitoring.manualControlEnabled := FALSE;
   sepaGripper.sequence.monitoring.manualModeChangeEnabled := FALSE;
   sepaGripper.sequence.monitoring.memoryStepTimer := 16#0000_4E92_AEA0_D6D2;
   jellyRollWinder.jobs.commands.setJobNumber := 0;
   jellyRollWinder.jobs.commands.reset := FALSE;
   jellyRollWinder.jobs.status.activeJobNumber := 0;
   jellyRollWinder.jobs.status.previousCycleJobNumber := 0;
   jellyRollWinder.jobs.status.manualControlEnabled := FALSE;
   jellyRollWinder.jobs.status.memoryJobTime := 16#0000_4E90_62D8_99E4;
   jellyRollWinder.sequence.commands.setAutomaticMode := FALSE;
   jellyRollWinder.sequence.commands.setSingleStepMode := FALSE;
   jellyRollWinder.sequence.commands.off := FALSE;
   jellyRollWinder.sequence.commands.initialize := FALSE;
   jellyRollWinder.sequence.commands.start := FALSE;
   jellyRollWinder.sequence.commands.immediateStop := FALSE;
   jellyRollWinder.sequence.commands.hold := FALSE;
   jellyRollWinder.sequence.commands.nextStep := FALSE;
   jellyRollWinder.sequence.commands.interlockStepChange := FALSE;
   jellyRollWinder.sequence.monitoring.automaticMode := TRUE;
   jellyRollWinder.sequence.monitoring.singleStepMode := FALSE;
   jellyRollWinder.sequence.monitoring.currentStep := 1;
   jellyRollWinder.sequence.monitoring.nextStep := 1;
   jellyRollWinder.sequence.monitoring.previousStep := 190;
   jellyRollWinder.sequence.monitoring.currentStepSTRING := 'N/A';
   jellyRollWinder.sequence.monitoring.nextStepSTRING := 'N/A';
   jellyRollWinder.sequence.monitoring.previousStepSTRING := 'N/A';
   jellyRollWinder.sequence.monitoring.inStepIdle := TRUE;
   jellyRollWinder.sequence.monitoring.inStepStopped := FALSE;
   jellyRollWinder.sequence.monitoring.seqActive := TRUE;
   jellyRollWinder.sequence.monitoring.stepActive := TRUE;
   jellyRollWinder.sequence.monitoring.stepComplete := FALSE;
   jellyRollWinder.sequence.monitoring.executionEnabled := TRUE;
   jellyRollWinder.sequence.monitoring.initRequired := FALSE;
   jellyRollWinder.sequence.monitoring.stepChangeReleased := TRUE;
   jellyRollWinder.sequence.monitoring.justSteppedPulse := FALSE;
   jellyRollWinder.sequence.monitoring.manualControlEnabled := FALSE;
   jellyRollWinder.sequence.monitoring.manualModeChangeEnabled := FALSE;
   jellyRollWinder.sequence.monitoring.memoryStepTimer := 16#0000_4E90_62D7_E3E5;
   distance.SepaClampToSepaGripperDisance.setValue.direction := FALSE;
   distance.SepaClampToSepaGripperDisance.setValue.distanceLimitSV := 0.0;
   distance.SepaClampToSepaGripperDisance.setValue.distancePTPSV := 0.0;
   distance.SepaClampToSepaGripperDisance.processValue.distanceOutPos := FALSE;
   distance.SepaClampToSepaGripperDisance.processValue.distanceLimitPV := 0.0;
   distance.SepaClampToSepaGripperDisance.processValue.currentDistance := -200.0;
   distance.SepaGripperToSepaClampDisance.setValue.direction := FALSE;
   distance.SepaGripperToSepaClampDisance.setValue.distanceLimitSV := 0.0;
   distance.SepaGripperToSepaClampDisance.setValue.distancePTPSV := 0.0;
   distance.SepaGripperToSepaClampDisance.processValue.distanceOutPos := FALSE;
   distance.SepaGripperToSepaClampDisance.processValue.distanceLimitPV := 0.0;
   distance.SepaGripperToSepaClampDisance.processValue.currentDistance := -200.0;
   distance.SepaGripperAxisCHomeDeg.setValue.direction := FALSE;
   distance.SepaGripperAxisCHomeDeg.setValue.distanceLimitSV := 0.0;
   distance.SepaGripperAxisCHomeDeg.setValue.distancePTPSV := 0.0;
   distance.SepaGripperAxisCHomeDeg.processValue.distanceOutPos := FALSE;
   distance.SepaGripperAxisCHomeDeg.processValue.distanceLimitPV := 0.0;
   distance.SepaGripperAxisCHomeDeg.processValue.currentDistance := 0.0;
   distance.SepaGripperAxisXHomeDis.setValue.direction := FALSE;
   distance.SepaGripperAxisXHomeDis.setValue.distanceLimitSV := 0.0;
   distance.SepaGripperAxisXHomeDis.setValue.distancePTPSV := 0.0;
   distance.SepaGripperAxisXHomeDis.processValue.distanceOutPos := FALSE;
   distance.SepaGripperAxisXHomeDis.processValue.distanceLimitPV := 0.0;
   distance.SepaGripperAxisXHomeDis.processValue.currentDistance := 0.0;
   cmSepaClampDetectSensor.commands.refreshConfiguration := FALSE;
   cmSepaClampDetectSensor.commands.editConfiguration := FALSE;
   cmSepaClampDetectSensor.commands.saveConfiguration := FALSE;
   cmSepaClampDetectSensor.commands.reset := FALSE;
   cmSepaClampDetectSensor.monitoring.enable := TRUE;
   cmSepaClampDetectSensor.monitoring.referenceDesignator := WSTRING#'DigitalSignal';
   cmSepaClampDetectSensor.monitoring.simulation := FALSE;
   cmSepaClampDetectSensor.monitoring.processValue := FALSE;
   cmSepaClampDetectSensor.monitoring.error := FALSE;
   cmSepaClampDetectSensor.monitoring.status := 16#0000;
   cmSepaClampDetectSensor.configuration.referenceDesignator := WSTRING#'DigitalSignal';
   cmSepaClampDetectSensor.configuration.onDelay := T#0MS;
   cmSepaClampDetectSensor.configuration.offDelay := T#0MS;
   cmSepaClampDetectSensor.configuration.default := FALSE;
   cmSepaClampDetectSensor.configuration.invertProcessValue := FALSE;
   cmSepaClampDetectSensor.configuration.disableAlarms := FALSE;
   cmSepaGripperDetectSensor.commands.refreshConfiguration := FALSE;
   cmSepaGripperDetectSensor.commands.editConfiguration := FALSE;
   cmSepaGripperDetectSensor.commands.saveConfiguration := FALSE;
   cmSepaGripperDetectSensor.commands.reset := FALSE;
   cmSepaGripperDetectSensor.monitoring.enable := TRUE;
   cmSepaGripperDetectSensor.monitoring.referenceDesignator := WSTRING#'DigitalSignal';
   cmSepaGripperDetectSensor.monitoring.simulation := FALSE;
   cmSepaGripperDetectSensor.monitoring.processValue := FALSE;
   cmSepaGripperDetectSensor.monitoring.error := FALSE;
   cmSepaGripperDetectSensor.monitoring.status := 16#0000;
   cmSepaGripperDetectSensor.configuration.referenceDesignator := WSTRING#'DigitalSignal';
   cmSepaGripperDetectSensor.configuration.onDelay := T#0MS;
   cmSepaGripperDetectSensor.configuration.offDelay := T#0MS;
   cmSepaGripperDetectSensor.configuration.default := FALSE;
   cmSepaGripperDetectSensor.configuration.invertProcessValue := FALSE;
   cmSepaGripperDetectSensor.configuration.disableAlarms := FALSE;
   cmJRWinderDetectSensor.commands.refreshConfiguration := FALSE;
   cmJRWinderDetectSensor.commands.editConfiguration := FALSE;
   cmJRWinderDetectSensor.commands.saveConfiguration := FALSE;
   cmJRWinderDetectSensor.commands.reset := FALSE;
   cmJRWinderDetectSensor.monitoring.enable := TRUE;
   cmJRWinderDetectSensor.monitoring.referenceDesignator := WSTRING#'DigitalSignal';
   cmJRWinderDetectSensor.monitoring.simulation := FALSE;
   cmJRWinderDetectSensor.monitoring.processValue := FALSE;
   cmJRWinderDetectSensor.monitoring.error := FALSE;
   cmJRWinderDetectSensor.monitoring.status := 16#0000;
   cmJRWinderDetectSensor.configuration.referenceDesignator := WSTRING#'DigitalSignal';
   cmJRWinderDetectSensor.configuration.onDelay := T#0MS;
   cmJRWinderDetectSensor.configuration.offDelay := T#0MS;
   cmJRWinderDetectSensor.configuration.default := FALSE;
   cmJRWinderDetectSensor.configuration.invertProcessValue := FALSE;
   cmJRWinderDetectSensor.configuration.disableAlarms := FALSE;
   cmSepaClampSafetyPinDetectSensor.commands.refreshConfiguration := FALSE;
   cmSepaClampSafetyPinDetectSensor.commands.editConfiguration := FALSE;
   cmSepaClampSafetyPinDetectSensor.commands.saveConfiguration := FALSE;
   cmSepaClampSafetyPinDetectSensor.commands.reset := FALSE;
   cmSepaClampSafetyPinDetectSensor.monitoring.enable := TRUE;
   cmSepaClampSafetyPinDetectSensor.monitoring.referenceDesignator := WSTRING#'DigitalSignal';
   cmSepaClampSafetyPinDetectSensor.monitoring.simulation := FALSE;
   cmSepaClampSafetyPinDetectSensor.monitoring.processValue := FALSE;
   cmSepaClampSafetyPinDetectSensor.monitoring.error := FALSE;
   cmSepaClampSafetyPinDetectSensor.monitoring.status := 16#0000;
   cmSepaClampSafetyPinDetectSensor.configuration.referenceDesignator := WSTRING#'DigitalSignal';
   cmSepaClampSafetyPinDetectSensor.configuration.onDelay := T#0MS;
   cmSepaClampSafetyPinDetectSensor.configuration.offDelay := T#0MS;
   cmSepaClampSafetyPinDetectSensor.configuration.default := FALSE;
   cmSepaClampSafetyPinDetectSensor.configuration.invertProcessValue := FALSE;
   cmSepaClampSafetyPinDetectSensor.configuration.disableAlarms := FALSE;
   cmSepaGripperSafetyPinDetectSensor.commands.refreshConfiguration := FALSE;
   cmSepaGripperSafetyPinDetectSensor.commands.editConfiguration := FALSE;
   cmSepaGripperSafetyPinDetectSensor.commands.saveConfiguration := FALSE;
   cmSepaGripperSafetyPinDetectSensor.commands.reset := FALSE;
   cmSepaGripperSafetyPinDetectSensor.monitoring.enable := TRUE;
   cmSepaGripperSafetyPinDetectSensor.monitoring.referenceDesignator := WSTRING#'DigitalSignal';
   cmSepaGripperSafetyPinDetectSensor.monitoring.simulation := FALSE;
   cmSepaGripperSafetyPinDetectSensor.monitoring.processValue := FALSE;
   cmSepaGripperSafetyPinDetectSensor.monitoring.error := FALSE;
   cmSepaGripperSafetyPinDetectSensor.monitoring.status := 16#0000;
   cmSepaGripperSafetyPinDetectSensor.configuration.referenceDesignator := WSTRING#'DigitalSignal';
   cmSepaGripperSafetyPinDetectSensor.configuration.onDelay := T#0MS;
   cmSepaGripperSafetyPinDetectSensor.configuration.offDelay := T#0MS;
   cmSepaGripperSafetyPinDetectSensor.configuration.default := FALSE;
   cmSepaGripperSafetyPinDetectSensor.configuration.invertProcessValue := FALSE;
   cmSepaGripperSafetyPinDetectSensor.configuration.disableAlarms := FALSE;
   cmSepaClampnCutterAxisX.commandConfiguration.generalSettings.stopOnError := TRUE;
   cmSepaClampnCutterAxisX.commandConfiguration.generalSettings.resetWithRestart := FALSE;
   cmSepaClampnCutterAxisX.commandConfiguration.generalSettings.abortWaitingSyncCmd := TRUE;
   cmSepaClampnCutterAxisX.commandConfiguration.power.startMode := 1;
   cmSepaClampnCutterAxisX.commandConfiguration.power.stopMode := 0;
   cmSepaClampnCutterAxisX.commandConfiguration.power.syncMotionSimulation := FALSE;
   cmSepaClampnCutterAxisX.commandConfiguration.power.syncMotionSimulationExtendedMode := -1;
   cmSepaClampnCutterAxisX.commandConfiguration.jog.velocity := 0.0;
   cmSepaClampnCutterAxisX.commandConfiguration.jog.acceleration := -1.0;
   cmSepaClampnCutterAxisX.commandConfiguration.jog.deceleration := -1.0;
   cmSepaClampnCutterAxisX.commandConfiguration.jog.jerk := -1.0;
   cmSepaClampnCutterAxisX.commandConfiguration.jog.positionControlled := TRUE;
   cmSepaClampnCutterAxisX.commandConfiguration.jog.increment := 0.0;
   cmSepaClampnCutterAxisX.commandConfiguration.jog.mode := 0;
   cmSepaClampnCutterAxisX.commandConfiguration.moveVelocity.velocity := 0.0;
   cmSepaClampnCutterAxisX.commandConfiguration.moveVelocity.acceleration := -1.0;
   cmSepaClampnCutterAxisX.commandConfiguration.moveVelocity.deceleration := -1.0;
   cmSepaClampnCutterAxisX.commandConfiguration.moveVelocity.jerk := -1.0;
   cmSepaClampnCutterAxisX.commandConfiguration.moveVelocity.direction := 0;
   cmSepaClampnCutterAxisX.commandConfiguration.moveVelocity.positionControlled := TRUE;
   cmSepaClampnCutterAxisX.commandConfiguration.moveVelocity.velocityChangeOnTheFly := FALSE;
   cmSepaClampnCutterAxisX.commandConfiguration.stop.deceleration := -1.0;
   cmSepaClampnCutterAxisX.commandConfiguration.stop.jerk := -1.0;
   cmSepaClampnCutterAxisX.commandConfiguration.stop.abortAcceleration := FALSE;
   cmSepaClampnCutterAxisX.commandConfiguration.fastStop.deceleration := -1.0;
   cmSepaClampnCutterAxisX.commandConfiguration.fastStop.jerk := -1.0;
   cmSepaClampnCutterAxisX.commandConfiguration.fastStop.abortAcceleration := FALSE;
   cmSepaClampnCutterAxisX.commandConfiguration.fastStop.replaceStopPossible := FALSE;
   cmSepaClampnCutterAxisX.commandConfiguration.torqueLimiting.limit := -1.0;
   cmSepaClampnCutterAxisX.commandConfiguration.torqueLimiting.mode := 0;
   cmSepaClampnCutterAxisX.commandConfiguration.homing.position := 0.0;
   cmSepaClampnCutterAxisX.commandConfiguration.homing.mode := 0;
   cmSepaClampnCutterAxisX.commandConfiguration.homing.sensor := 0;
   cmSepaClampnCutterAxisX.commandConfiguration.homing.extendedMode := -1;
   cmSepaClampnCutterAxisX.commandConfiguration.homing.extendedModeTorqueLimit := 0.0;
   cmSepaClampnCutterAxisX.commandConfiguration.homing.extendedModeTargetPosition := 0.0;
   cmSepaClampnCutterAxisX.commandConfiguration.posRelative.distance := 0.0;
   cmSepaClampnCutterAxisX.commandConfiguration.posRelative.velocity := -1.0;
   cmSepaClampnCutterAxisX.commandConfiguration.posRelative.acceleration := -1.0;
   cmSepaClampnCutterAxisX.commandConfiguration.posRelative.deceleration := -1.0;
   cmSepaClampnCutterAxisX.commandConfiguration.posRelative.jerk := -1.0;
   cmSepaClampnCutterAxisX.commandConfiguration.posRelative.direction := 0;
   cmSepaClampnCutterAxisX.commandConfiguration.posAbsolute.position := 0.0;
   cmSepaClampnCutterAxisX.commandConfiguration.posAbsolute.velocity := -1.0;
   cmSepaClampnCutterAxisX.commandConfiguration.posAbsolute.acceleration := -1.0;
   cmSepaClampnCutterAxisX.commandConfiguration.posAbsolute.deceleration := -1.0;
   cmSepaClampnCutterAxisX.commandConfiguration.posAbsolute.jerk := -1.0;
   cmSepaClampnCutterAxisX.commandConfiguration.posAbsolute.direction := 1;
   cmSepaClampnCutterAxisX.commandConfiguration.posAbsolute.positionChangeOnTheFly := FALSE;
   cmSepaClampnCutterAxisX.commandConfiguration.posAbsolute.velocityChangeOnTheFly := FALSE;
   cmSepaClampnCutterAxisX.commandConfiguration.posSuperimposed.distance := 0.0;
   cmSepaClampnCutterAxisX.commandConfiguration.posSuperimposed.velocityDiff := -1.0;
   cmSepaClampnCutterAxisX.commandConfiguration.posSuperimposed.acceleration := -1.0;
   cmSepaClampnCutterAxisX.commandConfiguration.posSuperimposed.deceleration := -1.0;
   cmSepaClampnCutterAxisX.commandConfiguration.posSuperimposed.jerk := -1.0;
   cmSepaClampnCutterAxisX.commandConfiguration.posSuperimposed.direction := 0;
   cmSepaClampnCutterAxisX.commandConfiguration.haltSuperimposed.deceleration := -1.0;
   cmSepaClampnCutterAxisX.commandConfiguration.haltSuperimposed.jerk := -1.0;
   cmSepaClampnCutterAxisX.commandConfiguration.haltSuperimposed.abortAcceleration := FALSE;
   cmSepaClampnCutterAxisX.commandConfiguration.gearInRelative.ratioNumerator := 1;
   cmSepaClampnCutterAxisX.commandConfiguration.gearInRelative.ratioDenominator := 1;
   cmSepaClampnCutterAxisX.commandConfiguration.gearInRelative.acceleration := -1.0;
   cmSepaClampnCutterAxisX.commandConfiguration.gearInRelative.deceleration := -1.0;
   cmSepaClampnCutterAxisX.commandConfiguration.gearInRelative.jerk := -1.0;
   cmSepaClampnCutterAxisX.commandConfiguration.gearInRelative.ratioChangeOnTheFly := FALSE;
   cmSepaClampnCutterAxisX.commandConfiguration.gearInAbsolute.ratioNumerator := 1;
   cmSepaClampnCutterAxisX.commandConfiguration.gearInAbsolute.ratioDenominator := 1;
   cmSepaClampnCutterAxisX.commandConfiguration.gearInAbsolute.masterSyncPosition := 0.0;
   cmSepaClampnCutterAxisX.commandConfiguration.gearInAbsolute.slaveSyncPosition := 0.0;
   cmSepaClampnCutterAxisX.commandConfiguration.gearInAbsolute.syncProfileReference := 1;
   cmSepaClampnCutterAxisX.commandConfiguration.gearInAbsolute.masterStartDistance := 0.0;
   cmSepaClampnCutterAxisX.commandConfiguration.gearInAbsolute.velocity := -1.0;
   cmSepaClampnCutterAxisX.commandConfiguration.gearInAbsolute.acceleration := -1.0;
   cmSepaClampnCutterAxisX.commandConfiguration.gearInAbsolute.deceleration := -1.0;
   cmSepaClampnCutterAxisX.commandConfiguration.gearInAbsolute.jerk := -1.0;
   cmSepaClampnCutterAxisX.commandConfiguration.gearInAbsolute.syncDirection := 1;
   cmSepaClampnCutterAxisX.commandConfiguration.gearInAbsolute.ratioChangeOnTheFly := FALSE;
   cmSepaClampnCutterAxisX.commandConfiguration.gearInVelocity.continuousUpdate := FALSE;
   cmSepaClampnCutterAxisX.commandConfiguration.gearInVelocity.ratioNumerator := 1;
   cmSepaClampnCutterAxisX.commandConfiguration.gearInVelocity.ratioDenominator := 1;
   cmSepaClampnCutterAxisX.commandConfiguration.gearInVelocity.acceleration := -1.0;
   cmSepaClampnCutterAxisX.commandConfiguration.gearInVelocity.deceleration := -1.0;
   cmSepaClampnCutterAxisX.commandConfiguration.gearInVelocity.jerk := -1.0;
   cmSepaClampnCutterAxisX.commandConfiguration.gearInVelocity.positionControlled := FALSE;
   cmSepaClampnCutterAxisX.commandConfiguration.camIn.masterOffset := 0.0;
   cmSepaClampnCutterAxisX.commandConfiguration.camIn.slaveOffset := 0.0;
   cmSepaClampnCutterAxisX.commandConfiguration.camIn.masterScaling := 1.0;
   cmSepaClampnCutterAxisX.commandConfiguration.camIn.slaveScaling := 1.0;
   cmSepaClampnCutterAxisX.commandConfiguration.camIn.masterSyncPosition := 0.0;
   cmSepaClampnCutterAxisX.commandConfiguration.camIn.syncProfileReference := 1;
   cmSepaClampnCutterAxisX.commandConfiguration.camIn.masterStartDistance := 0.0;
   cmSepaClampnCutterAxisX.commandConfiguration.camIn.velocity := -1.0;
   cmSepaClampnCutterAxisX.commandConfiguration.camIn.acceleration := -1.0;
   cmSepaClampnCutterAxisX.commandConfiguration.camIn.deceleration := -1.0;
   cmSepaClampnCutterAxisX.commandConfiguration.camIn.jerk := -1.0;
   cmSepaClampnCutterAxisX.commandConfiguration.camIn.applicationMode := 0;
   cmSepaClampnCutterAxisX.commandConfiguration.camIn.syncDirection := 1;
   cmSepaClampnCutterAxisX.commandConfiguration.gearOutCamOut.slavePosition := 0.0;
   cmSepaClampnCutterAxisX.commandConfiguration.gearOutCamOut.syncProfileReference := 1;
   cmSepaClampnCutterAxisX.commandConfiguration.gearOutCamOut.masterStopDistance := 0.0;
   cmSepaClampnCutterAxisX.commandConfiguration.gearOutCamOut.deceleration := -1.0;
   cmSepaClampnCutterAxisX.commandConfiguration.gearOutCamOut.jerk := -1.0;
   cmSepaClampnCutterAxisX.commandConfiguration.gearOutCamOut.syncOutDirection := 3;
   cmSepaClampnCutterAxisX.commandConfiguration.gearOutCamOut.gearOutCamOutMode := -1;
   cmSepaClampnCutterAxisX.commandConfiguration.phasing.phaseShift := 0.0;
   cmSepaClampnCutterAxisX.commandConfiguration.phasing.velocity := -1.0;
   cmSepaClampnCutterAxisX.commandConfiguration.phasing.acceleration := -1.0;
   cmSepaClampnCutterAxisX.commandConfiguration.phasing.deceleration := -1.0;
   cmSepaClampnCutterAxisX.commandConfiguration.phasing.jerk := -1.0;
   cmSepaClampnCutterAxisX.commandConfiguration.phasing.profileReference := 0;
   cmSepaClampnCutterAxisX.commandConfiguration.phasing.phasingDistance := 0.0;
   cmSepaClampnCutterAxisX.commandConfiguration.phasing.startPosition := 0.0;
   cmSepaClampnCutterAxisX.commandConfiguration.phasing.direction := 3;
   cmSepaClampnCutterAxisX.commandConfiguration.phasing.phaseAbsolute := TRUE;
   cmSepaClampnCutterAxisX.commandConfiguration.phasing.phaseShiftChangeOnTheFly := FALSE;
   cmSepaClampnCutterAxisX.commandConfiguration.offset.offset := 0.0;
   cmSepaClampnCutterAxisX.commandConfiguration.offset.profileReference := 1;
   cmSepaClampnCutterAxisX.commandConfiguration.offset.offsetDistance := 0.0;
   cmSepaClampnCutterAxisX.commandConfiguration.offset.startPosition := 0.0;
   cmSepaClampnCutterAxisX.commandConfiguration.offset.direction := 3;
   cmSepaClampnCutterAxisX.commandConfiguration.offset.offsetAbsolute := TRUE;
   cmSepaClampnCutterAxisX.commandConfiguration.offset.offsetChangeOnTheFly := FALSE;
   cmSepaClampnCutterAxisX.commands.enableMasterControl := TRUE;
   cmSepaClampnCutterAxisX.commands.enableAxis := FALSE;
   cmSepaClampnCutterAxisX.commands.resetAxis := FALSE;
   cmSepaClampnCutterAxisX.commands.openBrake := FALSE;
   cmSepaClampnCutterAxisX.commands.jogForward := FALSE;
   cmSepaClampnCutterAxisX.commands.jogBackward := FALSE;
   cmSepaClampnCutterAxisX.commands.moveVelocity := FALSE;
   cmSepaClampnCutterAxisX.commands.stop := FALSE;
   cmSepaClampnCutterAxisX.commands.fastStop := FALSE;
   cmSepaClampnCutterAxisX.commands.torqueLimiting := FALSE;
   cmSepaClampnCutterAxisX.commands.homing := FALSE;
   cmSepaClampnCutterAxisX.commands.posRelative := FALSE;
   cmSepaClampnCutterAxisX.commands.posAbsolute := FALSE;
   cmSepaClampnCutterAxisX.commands.posSuperimposed := FALSE;
   cmSepaClampnCutterAxisX.commands.haltSuperimposed := FALSE;
   cmSepaClampnCutterAxisX.commands.selectSetPosition := -1;
   cmSepaClampnCutterAxisX.commands.uploadParameters := FALSE;
   cmSepaClampnCutterAxisX.commands.refreshConfiguration := FALSE;
   cmSepaClampnCutterAxisX.commands.editConfiguration := FALSE;
   cmSepaClampnCutterAxisX.commands.saveConfiguration := FALSE;
   cmSepaClampnCutterAxisX.commands.uploadCurrentTorque := FALSE;
   cmSepaClampnCutterAxisX.commands.reset := FALSE;
   cmSepaClampnCutterAxisX.monitoring.enable := TRUE;
   cmSepaClampnCutterAxisX.monitoring.referenceDesignator := WSTRING#'SepaClampnCutterAxisX';
   cmSepaClampnCutterAxisX.monitoring.enabled := TRUE;
   cmSepaClampnCutterAxisX.monitoring.enableManualCmds := FALSE;
   cmSepaClampnCutterAxisX.monitoring.reset := FALSE;
   cmSepaClampnCutterAxisX.monitoring.resetAxis := FALSE;
   cmSepaClampnCutterAxisX.monitoring.enableAxis := TRUE;
   cmSepaClampnCutterAxisX.monitoring.openBrake := FALSE;
   cmSepaClampnCutterAxisX.monitoring.jogBackward := FALSE;
   cmSepaClampnCutterAxisX.monitoring.jogForward := FALSE;
   cmSepaClampnCutterAxisX.monitoring.moveVelocity := FALSE;
   cmSepaClampnCutterAxisX.monitoring.stop := FALSE;
   cmSepaClampnCutterAxisX.monitoring.fastStop := FALSE;
   cmSepaClampnCutterAxisX.monitoring.torqueLimiting := FALSE;
   cmSepaClampnCutterAxisX.monitoring.homing := FALSE;
   cmSepaClampnCutterAxisX.monitoring.posRelative := FALSE;
   cmSepaClampnCutterAxisX.monitoring.posAbsolute := FALSE;
   cmSepaClampnCutterAxisX.monitoring.posSuperimposed := FALSE;
   cmSepaClampnCutterAxisX.monitoring.haltSuperimposed := FALSE;
   cmSepaClampnCutterAxisX.monitoring.brakeOpened := FALSE;
   cmSepaClampnCutterAxisX.monitoring.axisEnabled := TRUE;
   cmSepaClampnCutterAxisX.monitoring.resetActive := FALSE;
   cmSepaClampnCutterAxisX.monitoring.inVelocity := FALSE;
   cmSepaClampnCutterAxisX.monitoring.inLimitation := FALSE;
   cmSepaClampnCutterAxisX.monitoring.inClamping := FALSE;
   cmSepaClampnCutterAxisX.monitoring.startSync := FALSE;
   cmSepaClampnCutterAxisX.monitoring.inSync := FALSE;
   cmSepaClampnCutterAxisX.monitoring.inSimulation := FALSE;
   cmSepaClampnCutterAxisX.monitoring.jogSelected := FALSE;
   cmSepaClampnCutterAxisX.monitoring.moveVelocitySelected := FALSE;
   cmSepaClampnCutterAxisX.monitoring.stopSelected := FALSE;
   cmSepaClampnCutterAxisX.monitoring.fastStopSelected := FALSE;
   cmSepaClampnCutterAxisX.monitoring.torqueLimitingSelected := FALSE;
   cmSepaClampnCutterAxisX.monitoring.homingSelected := FALSE;
   cmSepaClampnCutterAxisX.monitoring.posRelativeSelected := FALSE;
   cmSepaClampnCutterAxisX.monitoring.posAbsoluteSelected := FALSE;
   cmSepaClampnCutterAxisX.monitoring.posSuperimposedSelected := FALSE;
   cmSepaClampnCutterAxisX.monitoring.haltSuperimposedSelected := FALSE;
   cmSepaClampnCutterAxisX.monitoring.commandBusy := FALSE;
   cmSepaClampnCutterAxisX.monitoring.commandDone := FALSE;
   cmSepaClampnCutterAxisX.monitoring.commandAborted := FALSE;
   cmSepaClampnCutterAxisX.monitoring.homingCommandBusy := FALSE;
   cmSepaClampnCutterAxisX.monitoring.homingCommandDone := FALSE;
   cmSepaClampnCutterAxisX.monitoring.homingCommandAborted := FALSE;
   cmSepaClampnCutterAxisX.monitoring.superimposedBusy := FALSE;
   cmSepaClampnCutterAxisX.monitoring.superimposedDone := FALSE;
   cmSepaClampnCutterAxisX.monitoring.superimposedAborted := FALSE;
   cmSepaClampnCutterAxisX.monitoring.selectSetPosition := -1;
   cmSepaClampnCutterAxisX.monitoring.selectionController := FALSE;
   cmSepaClampnCutterAxisX.monitoring.interlockGeneral := TRUE;
   cmSepaClampnCutterAxisX.monitoring.interlockJogForward := TRUE;
   cmSepaClampnCutterAxisX.monitoring.interlockJogBackward := TRUE;
   cmSepaClampnCutterAxisX.monitoring.interlockWarningGeneral := FALSE;
   cmSepaClampnCutterAxisX.monitoring.interlockWarningJogForward := FALSE;
   cmSepaClampnCutterAxisX.monitoring.interlockWarningJogBackward := FALSE;
   cmSepaClampnCutterAxisX.monitoring.valid := TRUE;
   cmSepaClampnCutterAxisX.monitoring.busy := TRUE;
   cmSepaClampnCutterAxisX.monitoring.error := FALSE;
   cmSepaClampnCutterAxisX.monitoring.status := 16#7002;
   cmSepaClampnCutterAxisX.monitoring.subfunctionStatus := 16#0000;
   cmSepaClampnCutterAxisX.monitoring.actualPosition := 100.0;
   cmSepaClampnCutterAxisX.monitoring.actualSpeed := 0.0;
   cmSepaClampnCutterAxisX.monitoring.speedUnit := 1062;
   cmSepaClampnCutterAxisX.monitoring.positionUnit := 1013;
   cmSepaClampnCutterAxisX.monitoring.axisStatus1 := 16#0200_10E1;
   cmSepaClampnCutterAxisX.monitoring.axisStatus2 := 16#0000_0000;
   cmSepaClampnCutterAxisX.monitoring.axisType := 1;
   cmSepaClampnCutterAxisX.monitoring.maxVelocity := 2500.0;
   cmSepaClampnCutterAxisX.monitoring.actualCurrent := 0.0;
   cmSepaClampnCutterAxisX.monitoring.actualTorque := 0.0;
   cmSepaClampnCutterAxisX.monitoring.velocityOverrideEnabled := FALSE;
   cmSepaClampnCutterAxisX.monitoring.sinaParaError := FALSE;
   cmSepaClampnCutterAxisX.monitoring.sinaParaStatus := 16#0000_0000;
   cmSepaClampnCutterAxisX.configuration.referenceDesignator := WSTRING#'SepaClampnCutterAxisX';
   cmSepaClampnCutterAxisX.configuration.disableAlarms := FALSE;
   cmSepaClampnCutterAxisX.configuration.masterControlPopUp := TRUE;
   cmSepaClampnCutterAxisX.configuration.setPositions[0].position := 100.0;
   cmSepaClampnCutterAxisX.configuration.setPositions[1].position := 0.0;
   cmSepaClampnCutterAxisX.configuration.setPositions[2].position := 200.0;
   cmSepaClampnCutterAxisX.configuration.setPositions[3].position := 400.0;
   cmSepaClampnCutterAxisX.configuration.setPositions[4..15].position := 0.0;
   cmSepaClampnCutterAxisX.configuration.setPositions[0..3].velocity := 100.0;
   cmSepaClampnCutterAxisX.configuration.setPositions[4..15].velocity := -1.0;
   cmSepaClampnCutterAxisX.configuration.setPositions[0..3].acceleration := 1000.0;
   cmSepaClampnCutterAxisX.configuration.setPositions[4..15].acceleration := -1.0;
   cmSepaClampnCutterAxisX.configuration.setPositions[0..3].deceleration := 1000.0;
   cmSepaClampnCutterAxisX.configuration.setPositions[4..15].deceleration := -1.0;
   cmSepaClampnCutterAxisX.configuration.setPositions[0..15]."name" := '';
   cmSepaClampnCutterAxisZ.commandConfiguration.generalSettings.stopOnError := TRUE;
   cmSepaClampnCutterAxisZ.commandConfiguration.generalSettings.resetWithRestart := FALSE;
   cmSepaClampnCutterAxisZ.commandConfiguration.generalSettings.abortWaitingSyncCmd := TRUE;
   cmSepaClampnCutterAxisZ.commandConfiguration.power.startMode := 1;
   cmSepaClampnCutterAxisZ.commandConfiguration.power.stopMode := 0;
   cmSepaClampnCutterAxisZ.commandConfiguration.power.syncMotionSimulation := FALSE;
   cmSepaClampnCutterAxisZ.commandConfiguration.power.syncMotionSimulationExtendedMode := -1;
   cmSepaClampnCutterAxisZ.commandConfiguration.jog.velocity := 0.0;
   cmSepaClampnCutterAxisZ.commandConfiguration.jog.acceleration := -1.0;
   cmSepaClampnCutterAxisZ.commandConfiguration.jog.deceleration := -1.0;
   cmSepaClampnCutterAxisZ.commandConfiguration.jog.jerk := -1.0;
   cmSepaClampnCutterAxisZ.commandConfiguration.jog.positionControlled := TRUE;
   cmSepaClampnCutterAxisZ.commandConfiguration.jog.increment := 0.0;
   cmSepaClampnCutterAxisZ.commandConfiguration.jog.mode := 0;
   cmSepaClampnCutterAxisZ.commandConfiguration.moveVelocity.velocity := 0.0;
   cmSepaClampnCutterAxisZ.commandConfiguration.moveVelocity.acceleration := -1.0;
   cmSepaClampnCutterAxisZ.commandConfiguration.moveVelocity.deceleration := -1.0;
   cmSepaClampnCutterAxisZ.commandConfiguration.moveVelocity.jerk := -1.0;
   cmSepaClampnCutterAxisZ.commandConfiguration.moveVelocity.direction := 0;
   cmSepaClampnCutterAxisZ.commandConfiguration.moveVelocity.positionControlled := TRUE;
   cmSepaClampnCutterAxisZ.commandConfiguration.moveVelocity.velocityChangeOnTheFly := FALSE;
   cmSepaClampnCutterAxisZ.commandConfiguration.stop.deceleration := -1.0;
   cmSepaClampnCutterAxisZ.commandConfiguration.stop.jerk := -1.0;
   cmSepaClampnCutterAxisZ.commandConfiguration.stop.abortAcceleration := FALSE;
   cmSepaClampnCutterAxisZ.commandConfiguration.fastStop.deceleration := -1.0;
   cmSepaClampnCutterAxisZ.commandConfiguration.fastStop.jerk := -1.0;
   cmSepaClampnCutterAxisZ.commandConfiguration.fastStop.abortAcceleration := FALSE;
   cmSepaClampnCutterAxisZ.commandConfiguration.fastStop.replaceStopPossible := FALSE;
   cmSepaClampnCutterAxisZ.commandConfiguration.torqueLimiting.limit := -1.0;
   cmSepaClampnCutterAxisZ.commandConfiguration.torqueLimiting.mode := 0;
   cmSepaClampnCutterAxisZ.commandConfiguration.homing.position := 0.0;
   cmSepaClampnCutterAxisZ.commandConfiguration.homing.mode := 0;
   cmSepaClampnCutterAxisZ.commandConfiguration.homing.sensor := 0;
   cmSepaClampnCutterAxisZ.commandConfiguration.homing.extendedMode := -1;
   cmSepaClampnCutterAxisZ.commandConfiguration.homing.extendedModeTorqueLimit := 0.0;
   cmSepaClampnCutterAxisZ.commandConfiguration.homing.extendedModeTargetPosition := 0.0;
   cmSepaClampnCutterAxisZ.commandConfiguration.posRelative.distance := 0.0;
   cmSepaClampnCutterAxisZ.commandConfiguration.posRelative.velocity := -1.0;
   cmSepaClampnCutterAxisZ.commandConfiguration.posRelative.acceleration := -1.0;
   cmSepaClampnCutterAxisZ.commandConfiguration.posRelative.deceleration := -1.0;
   cmSepaClampnCutterAxisZ.commandConfiguration.posRelative.jerk := -1.0;
   cmSepaClampnCutterAxisZ.commandConfiguration.posRelative.direction := 0;
   cmSepaClampnCutterAxisZ.commandConfiguration.posAbsolute.position := 0.0;
   cmSepaClampnCutterAxisZ.commandConfiguration.posAbsolute.velocity := -1.0;
   cmSepaClampnCutterAxisZ.commandConfiguration.posAbsolute.acceleration := -1.0;
   cmSepaClampnCutterAxisZ.commandConfiguration.posAbsolute.deceleration := -1.0;
   cmSepaClampnCutterAxisZ.commandConfiguration.posAbsolute.jerk := -1.0;
   cmSepaClampnCutterAxisZ.commandConfiguration.posAbsolute.direction := 1;
   cmSepaClampnCutterAxisZ.commandConfiguration.posAbsolute.positionChangeOnTheFly := FALSE;
   cmSepaClampnCutterAxisZ.commandConfiguration.posAbsolute.velocityChangeOnTheFly := FALSE;
   cmSepaClampnCutterAxisZ.commandConfiguration.posSuperimposed.distance := 0.0;
   cmSepaClampnCutterAxisZ.commandConfiguration.posSuperimposed.velocityDiff := -1.0;
   cmSepaClampnCutterAxisZ.commandConfiguration.posSuperimposed.acceleration := -1.0;
   cmSepaClampnCutterAxisZ.commandConfiguration.posSuperimposed.deceleration := -1.0;
   cmSepaClampnCutterAxisZ.commandConfiguration.posSuperimposed.jerk := -1.0;
   cmSepaClampnCutterAxisZ.commandConfiguration.posSuperimposed.direction := 0;
   cmSepaClampnCutterAxisZ.commandConfiguration.haltSuperimposed.deceleration := -1.0;
   cmSepaClampnCutterAxisZ.commandConfiguration.haltSuperimposed.jerk := -1.0;
   cmSepaClampnCutterAxisZ.commandConfiguration.haltSuperimposed.abortAcceleration := FALSE;
   cmSepaClampnCutterAxisZ.commandConfiguration.gearInRelative.ratioNumerator := 1;
   cmSepaClampnCutterAxisZ.commandConfiguration.gearInRelative.ratioDenominator := 1;
   cmSepaClampnCutterAxisZ.commandConfiguration.gearInRelative.acceleration := -1.0;
   cmSepaClampnCutterAxisZ.commandConfiguration.gearInRelative.deceleration := -1.0;
   cmSepaClampnCutterAxisZ.commandConfiguration.gearInRelative.jerk := -1.0;
   cmSepaClampnCutterAxisZ.commandConfiguration.gearInRelative.ratioChangeOnTheFly := FALSE;
   cmSepaClampnCutterAxisZ.commandConfiguration.gearInAbsolute.ratioNumerator := 1;
   cmSepaClampnCutterAxisZ.commandConfiguration.gearInAbsolute.ratioDenominator := 1;
   cmSepaClampnCutterAxisZ.commandConfiguration.gearInAbsolute.masterSyncPosition := 0.0;
   cmSepaClampnCutterAxisZ.commandConfiguration.gearInAbsolute.slaveSyncPosition := 0.0;
   cmSepaClampnCutterAxisZ.commandConfiguration.gearInAbsolute.syncProfileReference := 1;
   cmSepaClampnCutterAxisZ.commandConfiguration.gearInAbsolute.masterStartDistance := 0.0;
   cmSepaClampnCutterAxisZ.commandConfiguration.gearInAbsolute.velocity := -1.0;
   cmSepaClampnCutterAxisZ.commandConfiguration.gearInAbsolute.acceleration := -1.0;
   cmSepaClampnCutterAxisZ.commandConfiguration.gearInAbsolute.deceleration := -1.0;
   cmSepaClampnCutterAxisZ.commandConfiguration.gearInAbsolute.jerk := -1.0;
   cmSepaClampnCutterAxisZ.commandConfiguration.gearInAbsolute.syncDirection := 1;
   cmSepaClampnCutterAxisZ.commandConfiguration.gearInAbsolute.ratioChangeOnTheFly := FALSE;
   cmSepaClampnCutterAxisZ.commandConfiguration.gearInVelocity.continuousUpdate := FALSE;
   cmSepaClampnCutterAxisZ.commandConfiguration.gearInVelocity.ratioNumerator := 1;
   cmSepaClampnCutterAxisZ.commandConfiguration.gearInVelocity.ratioDenominator := 1;
   cmSepaClampnCutterAxisZ.commandConfiguration.gearInVelocity.acceleration := -1.0;
   cmSepaClampnCutterAxisZ.commandConfiguration.gearInVelocity.deceleration := -1.0;
   cmSepaClampnCutterAxisZ.commandConfiguration.gearInVelocity.jerk := -1.0;
   cmSepaClampnCutterAxisZ.commandConfiguration.gearInVelocity.positionControlled := FALSE;
   cmSepaClampnCutterAxisZ.commandConfiguration.camIn.masterOffset := 0.0;
   cmSepaClampnCutterAxisZ.commandConfiguration.camIn.slaveOffset := 0.0;
   cmSepaClampnCutterAxisZ.commandConfiguration.camIn.masterScaling := 1.0;
   cmSepaClampnCutterAxisZ.commandConfiguration.camIn.slaveScaling := 1.0;
   cmSepaClampnCutterAxisZ.commandConfiguration.camIn.masterSyncPosition := 0.0;
   cmSepaClampnCutterAxisZ.commandConfiguration.camIn.syncProfileReference := 1;
   cmSepaClampnCutterAxisZ.commandConfiguration.camIn.masterStartDistance := 0.0;
   cmSepaClampnCutterAxisZ.commandConfiguration.camIn.velocity := -1.0;
   cmSepaClampnCutterAxisZ.commandConfiguration.camIn.acceleration := -1.0;
   cmSepaClampnCutterAxisZ.commandConfiguration.camIn.deceleration := -1.0;
   cmSepaClampnCutterAxisZ.commandConfiguration.camIn.jerk := -1.0;
   cmSepaClampnCutterAxisZ.commandConfiguration.camIn.applicationMode := 0;
   cmSepaClampnCutterAxisZ.commandConfiguration.camIn.syncDirection := 1;
   cmSepaClampnCutterAxisZ.commandConfiguration.gearOutCamOut.slavePosition := 0.0;
   cmSepaClampnCutterAxisZ.commandConfiguration.gearOutCamOut.syncProfileReference := 0;
   cmSepaClampnCutterAxisZ.commandConfiguration.gearOutCamOut.masterStopDistance := 0.0;
   cmSepaClampnCutterAxisZ.commandConfiguration.gearOutCamOut.deceleration := -1.0;
   cmSepaClampnCutterAxisZ.commandConfiguration.gearOutCamOut.jerk := -1.0;
   cmSepaClampnCutterAxisZ.commandConfiguration.gearOutCamOut.syncOutDirection := 3;
   cmSepaClampnCutterAxisZ.commandConfiguration.gearOutCamOut.gearOutCamOutMode := -1;
   cmSepaClampnCutterAxisZ.commandConfiguration.phasing.phaseShift := 0.0;
   cmSepaClampnCutterAxisZ.commandConfiguration.phasing.velocity := -1.0;
   cmSepaClampnCutterAxisZ.commandConfiguration.phasing.acceleration := -1.0;
   cmSepaClampnCutterAxisZ.commandConfiguration.phasing.deceleration := -1.0;
   cmSepaClampnCutterAxisZ.commandConfiguration.phasing.jerk := -1.0;
   cmSepaClampnCutterAxisZ.commandConfiguration.phasing.profileReference := 0;
   cmSepaClampnCutterAxisZ.commandConfiguration.phasing.phasingDistance := 0.0;
   cmSepaClampnCutterAxisZ.commandConfiguration.phasing.startPosition := 0.0;
   cmSepaClampnCutterAxisZ.commandConfiguration.phasing.direction := 3;
   cmSepaClampnCutterAxisZ.commandConfiguration.phasing.phaseAbsolute := TRUE;
   cmSepaClampnCutterAxisZ.commandConfiguration.phasing.phaseShiftChangeOnTheFly := FALSE;
   cmSepaClampnCutterAxisZ.commandConfiguration.offset.offset := 0.0;
   cmSepaClampnCutterAxisZ.commandConfiguration.offset.profileReference := 1;
   cmSepaClampnCutterAxisZ.commandConfiguration.offset.offsetDistance := 0.0;
   cmSepaClampnCutterAxisZ.commandConfiguration.offset.startPosition := 0.0;
   cmSepaClampnCutterAxisZ.commandConfiguration.offset.direction := 3;
   cmSepaClampnCutterAxisZ.commandConfiguration.offset.offsetAbsolute := TRUE;
   cmSepaClampnCutterAxisZ.commandConfiguration.offset.offsetChangeOnTheFly := FALSE;
   cmSepaClampnCutterAxisZ.commands.enableMasterControl := TRUE;
   cmSepaClampnCutterAxisZ.commands.enableAxis := FALSE;
   cmSepaClampnCutterAxisZ.commands.resetAxis := FALSE;
   cmSepaClampnCutterAxisZ.commands.openBrake := FALSE;
   cmSepaClampnCutterAxisZ.commands.jogForward := FALSE;
   cmSepaClampnCutterAxisZ.commands.jogBackward := FALSE;
   cmSepaClampnCutterAxisZ.commands.moveVelocity := FALSE;
   cmSepaClampnCutterAxisZ.commands.stop := FALSE;
   cmSepaClampnCutterAxisZ.commands.fastStop := FALSE;
   cmSepaClampnCutterAxisZ.commands.torqueLimiting := FALSE;
   cmSepaClampnCutterAxisZ.commands.homing := FALSE;
   cmSepaClampnCutterAxisZ.commands.posRelative := FALSE;
   cmSepaClampnCutterAxisZ.commands.posAbsolute := FALSE;
   cmSepaClampnCutterAxisZ.commands.posSuperimposed := FALSE;
   cmSepaClampnCutterAxisZ.commands.haltSuperimposed := FALSE;
   cmSepaClampnCutterAxisZ.commands.selectSetPosition := -1;
   cmSepaClampnCutterAxisZ.commands.uploadParameters := FALSE;
   cmSepaClampnCutterAxisZ.commands.refreshConfiguration := FALSE;
   cmSepaClampnCutterAxisZ.commands.editConfiguration := FALSE;
   cmSepaClampnCutterAxisZ.commands.saveConfiguration := FALSE;
   cmSepaClampnCutterAxisZ.commands.uploadCurrentTorque := FALSE;
   cmSepaClampnCutterAxisZ.commands.reset := FALSE;
   cmSepaClampnCutterAxisZ.monitoring.enable := TRUE;
   cmSepaClampnCutterAxisZ.monitoring.referenceDesignator := WSTRING#'SepaClampnCutterAxisZ';
   cmSepaClampnCutterAxisZ.monitoring.enabled := TRUE;
   cmSepaClampnCutterAxisZ.monitoring.enableManualCmds := FALSE;
   cmSepaClampnCutterAxisZ.monitoring.reset := FALSE;
   cmSepaClampnCutterAxisZ.monitoring.resetAxis := FALSE;
   cmSepaClampnCutterAxisZ.monitoring.enableAxis := TRUE;
   cmSepaClampnCutterAxisZ.monitoring.openBrake := FALSE;
   cmSepaClampnCutterAxisZ.monitoring.jogBackward := FALSE;
   cmSepaClampnCutterAxisZ.monitoring.jogForward := FALSE;
   cmSepaClampnCutterAxisZ.monitoring.moveVelocity := FALSE;
   cmSepaClampnCutterAxisZ.monitoring.stop := FALSE;
   cmSepaClampnCutterAxisZ.monitoring.fastStop := FALSE;
   cmSepaClampnCutterAxisZ.monitoring.torqueLimiting := FALSE;
   cmSepaClampnCutterAxisZ.monitoring.homing := FALSE;
   cmSepaClampnCutterAxisZ.monitoring.posRelative := FALSE;
   cmSepaClampnCutterAxisZ.monitoring.posAbsolute := FALSE;
   cmSepaClampnCutterAxisZ.monitoring.posSuperimposed := FALSE;
   cmSepaClampnCutterAxisZ.monitoring.haltSuperimposed := FALSE;
   cmSepaClampnCutterAxisZ.monitoring.brakeOpened := FALSE;
   cmSepaClampnCutterAxisZ.monitoring.axisEnabled := TRUE;
   cmSepaClampnCutterAxisZ.monitoring.resetActive := FALSE;
   cmSepaClampnCutterAxisZ.monitoring.inVelocity := FALSE;
   cmSepaClampnCutterAxisZ.monitoring.inLimitation := FALSE;
   cmSepaClampnCutterAxisZ.monitoring.inClamping := FALSE;
   cmSepaClampnCutterAxisZ.monitoring.startSync := FALSE;
   cmSepaClampnCutterAxisZ.monitoring.inSync := FALSE;
   cmSepaClampnCutterAxisZ.monitoring.inSimulation := FALSE;
   cmSepaClampnCutterAxisZ.monitoring.jogSelected := FALSE;
   cmSepaClampnCutterAxisZ.monitoring.moveVelocitySelected := FALSE;
   cmSepaClampnCutterAxisZ.monitoring.stopSelected := FALSE;
   cmSepaClampnCutterAxisZ.monitoring.fastStopSelected := FALSE;
   cmSepaClampnCutterAxisZ.monitoring.torqueLimitingSelected := FALSE;
   cmSepaClampnCutterAxisZ.monitoring.homingSelected := FALSE;
   cmSepaClampnCutterAxisZ.monitoring.posRelativeSelected := FALSE;
   cmSepaClampnCutterAxisZ.monitoring.posAbsoluteSelected := FALSE;
   cmSepaClampnCutterAxisZ.monitoring.posSuperimposedSelected := FALSE;
   cmSepaClampnCutterAxisZ.monitoring.haltSuperimposedSelected := FALSE;
   cmSepaClampnCutterAxisZ.monitoring.commandBusy := FALSE;
   cmSepaClampnCutterAxisZ.monitoring.commandDone := FALSE;
   cmSepaClampnCutterAxisZ.monitoring.commandAborted := FALSE;
   cmSepaClampnCutterAxisZ.monitoring.homingCommandBusy := FALSE;
   cmSepaClampnCutterAxisZ.monitoring.homingCommandDone := FALSE;
   cmSepaClampnCutterAxisZ.monitoring.homingCommandAborted := FALSE;
   cmSepaClampnCutterAxisZ.monitoring.superimposedBusy := FALSE;
   cmSepaClampnCutterAxisZ.monitoring.superimposedDone := FALSE;
   cmSepaClampnCutterAxisZ.monitoring.superimposedAborted := FALSE;
   cmSepaClampnCutterAxisZ.monitoring.selectSetPosition := -1;
   cmSepaClampnCutterAxisZ.monitoring.selectionController := FALSE;
   cmSepaClampnCutterAxisZ.monitoring.interlockGeneral := TRUE;
   cmSepaClampnCutterAxisZ.monitoring.interlockJogForward := TRUE;
   cmSepaClampnCutterAxisZ.monitoring.interlockJogBackward := TRUE;
   cmSepaClampnCutterAxisZ.monitoring.interlockWarningGeneral := FALSE;
   cmSepaClampnCutterAxisZ.monitoring.interlockWarningJogForward := FALSE;
   cmSepaClampnCutterAxisZ.monitoring.interlockWarningJogBackward := FALSE;
   cmSepaClampnCutterAxisZ.monitoring.valid := TRUE;
   cmSepaClampnCutterAxisZ.monitoring.busy := TRUE;
   cmSepaClampnCutterAxisZ.monitoring.error := FALSE;
   cmSepaClampnCutterAxisZ.monitoring.status := 16#7002;
   cmSepaClampnCutterAxisZ.monitoring.subfunctionStatus := 16#0000;
   cmSepaClampnCutterAxisZ.monitoring.actualPosition := 0.0;
   cmSepaClampnCutterAxisZ.monitoring.actualSpeed := 0.0;
   cmSepaClampnCutterAxisZ.monitoring.speedUnit := 1062;
   cmSepaClampnCutterAxisZ.monitoring.positionUnit := 1013;
   cmSepaClampnCutterAxisZ.monitoring.axisStatus1 := 16#0200_10E1;
   cmSepaClampnCutterAxisZ.monitoring.axisStatus2 := 16#0000_0000;
   cmSepaClampnCutterAxisZ.monitoring.axisType := 1;
   cmSepaClampnCutterAxisZ.monitoring.maxVelocity := 2500.0;
   cmSepaClampnCutterAxisZ.monitoring.actualCurrent := 0.0;
   cmSepaClampnCutterAxisZ.monitoring.actualTorque := 0.0;
   cmSepaClampnCutterAxisZ.monitoring.velocityOverrideEnabled := FALSE;
   cmSepaClampnCutterAxisZ.monitoring.sinaParaError := FALSE;
   cmSepaClampnCutterAxisZ.monitoring.sinaParaStatus := 16#0000_0000;
   cmSepaClampnCutterAxisZ.configuration.referenceDesignator := WSTRING#'SepaClampnCutterAxisZ';
   cmSepaClampnCutterAxisZ.configuration.disableAlarms := FALSE;
   cmSepaClampnCutterAxisZ.configuration.masterControlPopUp := TRUE;
   cmSepaClampnCutterAxisZ.configuration.setPositions[0].position := 0.0;
   cmSepaClampnCutterAxisZ.configuration.setPositions[1].position := 25.0;
   cmSepaClampnCutterAxisZ.configuration.setPositions[2].position := 50.0;
   cmSepaClampnCutterAxisZ.configuration.setPositions[3..15].position := 0.0;
   cmSepaClampnCutterAxisZ.configuration.setPositions[0..2].velocity := 50.0;
   cmSepaClampnCutterAxisZ.configuration.setPositions[3..15].velocity := -1.0;
   cmSepaClampnCutterAxisZ.configuration.setPositions[0..2].acceleration := 500.0;
   cmSepaClampnCutterAxisZ.configuration.setPositions[3..15].acceleration := -1.0;
   cmSepaClampnCutterAxisZ.configuration.setPositions[0..2].deceleration := 500.0;
   cmSepaClampnCutterAxisZ.configuration.setPositions[3..15].deceleration := -1.0;
   cmSepaClampnCutterAxisZ.configuration.setPositions[0..15]."name" := '';
   cmSepaGripperAxisX.commandConfiguration.generalSettings.stopOnError := TRUE;
   cmSepaGripperAxisX.commandConfiguration.generalSettings.resetWithRestart := FALSE;
   cmSepaGripperAxisX.commandConfiguration.generalSettings.abortWaitingSyncCmd := TRUE;
   cmSepaGripperAxisX.commandConfiguration.power.startMode := 1;
   cmSepaGripperAxisX.commandConfiguration.power.stopMode := 0;
   cmSepaGripperAxisX.commandConfiguration.power.syncMotionSimulation := FALSE;
   cmSepaGripperAxisX.commandConfiguration.power.syncMotionSimulationExtendedMode := -1;
   cmSepaGripperAxisX.commandConfiguration.jog.velocity := 0.0;
   cmSepaGripperAxisX.commandConfiguration.jog.acceleration := -1.0;
   cmSepaGripperAxisX.commandConfiguration.jog.deceleration := -1.0;
   cmSepaGripperAxisX.commandConfiguration.jog.jerk := -1.0;
   cmSepaGripperAxisX.commandConfiguration.jog.positionControlled := TRUE;
   cmSepaGripperAxisX.commandConfiguration.jog.increment := 0.0;
   cmSepaGripperAxisX.commandConfiguration.jog.mode := 0;
   cmSepaGripperAxisX.commandConfiguration.moveVelocity.velocity := 0.0;
   cmSepaGripperAxisX.commandConfiguration.moveVelocity.acceleration := -1.0;
   cmSepaGripperAxisX.commandConfiguration.moveVelocity.deceleration := -1.0;
   cmSepaGripperAxisX.commandConfiguration.moveVelocity.jerk := -1.0;
   cmSepaGripperAxisX.commandConfiguration.moveVelocity.direction := 0;
   cmSepaGripperAxisX.commandConfiguration.moveVelocity.positionControlled := TRUE;
   cmSepaGripperAxisX.commandConfiguration.moveVelocity.velocityChangeOnTheFly := FALSE;
   cmSepaGripperAxisX.commandConfiguration.stop.deceleration := -1.0;
   cmSepaGripperAxisX.commandConfiguration.stop.jerk := -1.0;
   cmSepaGripperAxisX.commandConfiguration.stop.abortAcceleration := FALSE;
   cmSepaGripperAxisX.commandConfiguration.fastStop.deceleration := -1.0;
   cmSepaGripperAxisX.commandConfiguration.fastStop.jerk := -1.0;
   cmSepaGripperAxisX.commandConfiguration.fastStop.abortAcceleration := FALSE;
   cmSepaGripperAxisX.commandConfiguration.fastStop.replaceStopPossible := FALSE;
   cmSepaGripperAxisX.commandConfiguration.torqueLimiting.limit := -1.0;
   cmSepaGripperAxisX.commandConfiguration.torqueLimiting.mode := 0;
   cmSepaGripperAxisX.commandConfiguration.homing.position := 0.0;
   cmSepaGripperAxisX.commandConfiguration.homing.mode := 0;
   cmSepaGripperAxisX.commandConfiguration.homing.sensor := 0;
   cmSepaGripperAxisX.commandConfiguration.homing.extendedMode := -1;
   cmSepaGripperAxisX.commandConfiguration.homing.extendedModeTorqueLimit := 0.0;
   cmSepaGripperAxisX.commandConfiguration.homing.extendedModeTargetPosition := 0.0;
   cmSepaGripperAxisX.commandConfiguration.posRelative.distance := 0.0;
   cmSepaGripperAxisX.commandConfiguration.posRelative.velocity := -1.0;
   cmSepaGripperAxisX.commandConfiguration.posRelative.acceleration := -1.0;
   cmSepaGripperAxisX.commandConfiguration.posRelative.deceleration := -1.0;
   cmSepaGripperAxisX.commandConfiguration.posRelative.jerk := -1.0;
   cmSepaGripperAxisX.commandConfiguration.posRelative.direction := 0;
   cmSepaGripperAxisX.commandConfiguration.posAbsolute.position := 27.5;
   cmSepaGripperAxisX.commandConfiguration.posAbsolute.velocity := 30.0;
   cmSepaGripperAxisX.commandConfiguration.posAbsolute.acceleration := 30.0;
   cmSepaGripperAxisX.commandConfiguration.posAbsolute.deceleration := 30.0;
   cmSepaGripperAxisX.commandConfiguration.posAbsolute.jerk := -1.0;
   cmSepaGripperAxisX.commandConfiguration.posAbsolute.direction := 1;
   cmSepaGripperAxisX.commandConfiguration.posAbsolute.positionChangeOnTheFly := FALSE;
   cmSepaGripperAxisX.commandConfiguration.posAbsolute.velocityChangeOnTheFly := FALSE;
   cmSepaGripperAxisX.commandConfiguration.posSuperimposed.distance := 0.0;
   cmSepaGripperAxisX.commandConfiguration.posSuperimposed.velocityDiff := -1.0;
   cmSepaGripperAxisX.commandConfiguration.posSuperimposed.acceleration := -1.0;
   cmSepaGripperAxisX.commandConfiguration.posSuperimposed.deceleration := -1.0;
   cmSepaGripperAxisX.commandConfiguration.posSuperimposed.jerk := -1.0;
   cmSepaGripperAxisX.commandConfiguration.posSuperimposed.direction := 0;
   cmSepaGripperAxisX.commandConfiguration.haltSuperimposed.deceleration := -1.0;
   cmSepaGripperAxisX.commandConfiguration.haltSuperimposed.jerk := -1.0;
   cmSepaGripperAxisX.commandConfiguration.haltSuperimposed.abortAcceleration := FALSE;
   cmSepaGripperAxisX.commandConfiguration.gearInRelative.ratioNumerator := 1;
   cmSepaGripperAxisX.commandConfiguration.gearInRelative.ratioDenominator := 1;
   cmSepaGripperAxisX.commandConfiguration.gearInRelative.acceleration := -1.0;
   cmSepaGripperAxisX.commandConfiguration.gearInRelative.deceleration := -1.0;
   cmSepaGripperAxisX.commandConfiguration.gearInRelative.jerk := -1.0;
   cmSepaGripperAxisX.commandConfiguration.gearInRelative.ratioChangeOnTheFly := FALSE;
   cmSepaGripperAxisX.commandConfiguration.gearInAbsolute.ratioNumerator := 1;
   cmSepaGripperAxisX.commandConfiguration.gearInAbsolute.ratioDenominator := 1;
   cmSepaGripperAxisX.commandConfiguration.gearInAbsolute.masterSyncPosition := 0.0;
   cmSepaGripperAxisX.commandConfiguration.gearInAbsolute.slaveSyncPosition := 0.0;
   cmSepaGripperAxisX.commandConfiguration.gearInAbsolute.syncProfileReference := 1;
   cmSepaGripperAxisX.commandConfiguration.gearInAbsolute.masterStartDistance := 0.0;
   cmSepaGripperAxisX.commandConfiguration.gearInAbsolute.velocity := -1.0;
   cmSepaGripperAxisX.commandConfiguration.gearInAbsolute.acceleration := -1.0;
   cmSepaGripperAxisX.commandConfiguration.gearInAbsolute.deceleration := -1.0;
   cmSepaGripperAxisX.commandConfiguration.gearInAbsolute.jerk := -1.0;
   cmSepaGripperAxisX.commandConfiguration.gearInAbsolute.syncDirection := 1;
   cmSepaGripperAxisX.commandConfiguration.gearInAbsolute.ratioChangeOnTheFly := FALSE;
   cmSepaGripperAxisX.commandConfiguration.gearInVelocity.continuousUpdate := FALSE;
   cmSepaGripperAxisX.commandConfiguration.gearInVelocity.ratioNumerator := 1;
   cmSepaGripperAxisX.commandConfiguration.gearInVelocity.ratioDenominator := 1;
   cmSepaGripperAxisX.commandConfiguration.gearInVelocity.acceleration := -1.0;
   cmSepaGripperAxisX.commandConfiguration.gearInVelocity.deceleration := -1.0;
   cmSepaGripperAxisX.commandConfiguration.gearInVelocity.jerk := -1.0;
   cmSepaGripperAxisX.commandConfiguration.gearInVelocity.positionControlled := FALSE;
   cmSepaGripperAxisX.commandConfiguration.camIn.masterOffset := 0.0;
   cmSepaGripperAxisX.commandConfiguration.camIn.slaveOffset := 0.0;
   cmSepaGripperAxisX.commandConfiguration.camIn.masterScaling := 1.0;
   cmSepaGripperAxisX.commandConfiguration.camIn.slaveScaling := 1.0;
   cmSepaGripperAxisX.commandConfiguration.camIn.masterSyncPosition := 0.0;
   cmSepaGripperAxisX.commandConfiguration.camIn.syncProfileReference := 1;
   cmSepaGripperAxisX.commandConfiguration.camIn.masterStartDistance := 0.0;
   cmSepaGripperAxisX.commandConfiguration.camIn.velocity := -1.0;
   cmSepaGripperAxisX.commandConfiguration.camIn.acceleration := -1.0;
   cmSepaGripperAxisX.commandConfiguration.camIn.deceleration := -1.0;
   cmSepaGripperAxisX.commandConfiguration.camIn.jerk := -1.0;
   cmSepaGripperAxisX.commandConfiguration.camIn.applicationMode := 0;
   cmSepaGripperAxisX.commandConfiguration.camIn.syncDirection := 1;
   cmSepaGripperAxisX.commandConfiguration.gearOutCamOut.slavePosition := 0.0;
   cmSepaGripperAxisX.commandConfiguration.gearOutCamOut.syncProfileReference := 1;
   cmSepaGripperAxisX.commandConfiguration.gearOutCamOut.masterStopDistance := 0.0;
   cmSepaGripperAxisX.commandConfiguration.gearOutCamOut.deceleration := -1.0;
   cmSepaGripperAxisX.commandConfiguration.gearOutCamOut.jerk := -1.0;
   cmSepaGripperAxisX.commandConfiguration.gearOutCamOut.syncOutDirection := 3;
   cmSepaGripperAxisX.commandConfiguration.gearOutCamOut.gearOutCamOutMode := -1;
   cmSepaGripperAxisX.commandConfiguration.phasing.phaseShift := 0.0;
   cmSepaGripperAxisX.commandConfiguration.phasing.velocity := -1.0;
   cmSepaGripperAxisX.commandConfiguration.phasing.acceleration := -1.0;
   cmSepaGripperAxisX.commandConfiguration.phasing.deceleration := -1.0;
   cmSepaGripperAxisX.commandConfiguration.phasing.jerk := -1.0;
   cmSepaGripperAxisX.commandConfiguration.phasing.profileReference := 0;
   cmSepaGripperAxisX.commandConfiguration.phasing.phasingDistance := 0.0;
   cmSepaGripperAxisX.commandConfiguration.phasing.startPosition := 0.0;
   cmSepaGripperAxisX.commandConfiguration.phasing.direction := 3;
   cmSepaGripperAxisX.commandConfiguration.phasing.phaseAbsolute := TRUE;
   cmSepaGripperAxisX.commandConfiguration.phasing.phaseShiftChangeOnTheFly := FALSE;
   cmSepaGripperAxisX.commandConfiguration.offset.offset := 0.0;
   cmSepaGripperAxisX.commandConfiguration.offset.profileReference := 1;
   cmSepaGripperAxisX.commandConfiguration.offset.offsetDistance := 0.0;
   cmSepaGripperAxisX.commandConfiguration.offset.startPosition := 0.0;
   cmSepaGripperAxisX.commandConfiguration.offset.direction := 3;
   cmSepaGripperAxisX.commandConfiguration.offset.offsetAbsolute := TRUE;
   cmSepaGripperAxisX.commandConfiguration.offset.offsetChangeOnTheFly := FALSE;
   cmSepaGripperAxisX.commands.enableMasterControl := TRUE;
   cmSepaGripperAxisX.commands.enableAxis := FALSE;
   cmSepaGripperAxisX.commands.resetAxis := FALSE;
   cmSepaGripperAxisX.commands.openBrake := FALSE;
   cmSepaGripperAxisX.commands.jogForward := FALSE;
   cmSepaGripperAxisX.commands.jogBackward := FALSE;
   cmSepaGripperAxisX.commands.moveVelocity := FALSE;
   cmSepaGripperAxisX.commands.stop := FALSE;
   cmSepaGripperAxisX.commands.fastStop := FALSE;
   cmSepaGripperAxisX.commands.torqueLimiting := FALSE;
   cmSepaGripperAxisX.commands.homing := FALSE;
   cmSepaGripperAxisX.commands.posRelative := FALSE;
   cmSepaGripperAxisX.commands.posAbsolute := FALSE;
   cmSepaGripperAxisX.commands.posSuperimposed := FALSE;
   cmSepaGripperAxisX.commands.haltSuperimposed := FALSE;
   cmSepaGripperAxisX.commands.selectSetPosition := -1;
   cmSepaGripperAxisX.commands.uploadParameters := FALSE;
   cmSepaGripperAxisX.commands.refreshConfiguration := FALSE;
   cmSepaGripperAxisX.commands.editConfiguration := FALSE;
   cmSepaGripperAxisX.commands.saveConfiguration := FALSE;
   cmSepaGripperAxisX.commands.uploadCurrentTorque := FALSE;
   cmSepaGripperAxisX.commands.reset := FALSE;
   cmSepaGripperAxisX.monitoring.enable := TRUE;
   cmSepaGripperAxisX.monitoring.referenceDesignator := WSTRING#'SepaGripperAxisX';
   cmSepaGripperAxisX.monitoring.enabled := TRUE;
   cmSepaGripperAxisX.monitoring.enableManualCmds := FALSE;
   cmSepaGripperAxisX.monitoring.reset := FALSE;
   cmSepaGripperAxisX.monitoring.resetAxis := FALSE;
   cmSepaGripperAxisX.monitoring.enableAxis := TRUE;
   cmSepaGripperAxisX.monitoring.openBrake := FALSE;
   cmSepaGripperAxisX.monitoring.jogBackward := FALSE;
   cmSepaGripperAxisX.monitoring.jogForward := FALSE;
   cmSepaGripperAxisX.monitoring.moveVelocity := FALSE;
   cmSepaGripperAxisX.monitoring.stop := FALSE;
   cmSepaGripperAxisX.monitoring.fastStop := FALSE;
   cmSepaGripperAxisX.monitoring.torqueLimiting := FALSE;
   cmSepaGripperAxisX.monitoring.homing := FALSE;
   cmSepaGripperAxisX.monitoring.posRelative := FALSE;
   cmSepaGripperAxisX.monitoring.posAbsolute := FALSE;
   cmSepaGripperAxisX.monitoring.posSuperimposed := FALSE;
   cmSepaGripperAxisX.monitoring.haltSuperimposed := FALSE;
   cmSepaGripperAxisX.monitoring.brakeOpened := FALSE;
   cmSepaGripperAxisX.monitoring.axisEnabled := TRUE;
   cmSepaGripperAxisX.monitoring.resetActive := FALSE;
   cmSepaGripperAxisX.monitoring.inVelocity := FALSE;
   cmSepaGripperAxisX.monitoring.inLimitation := FALSE;
   cmSepaGripperAxisX.monitoring.inClamping := FALSE;
   cmSepaGripperAxisX.monitoring.startSync := FALSE;
   cmSepaGripperAxisX.monitoring.inSync := FALSE;
   cmSepaGripperAxisX.monitoring.inSimulation := FALSE;
   cmSepaGripperAxisX.monitoring.jogSelected := FALSE;
   cmSepaGripperAxisX.monitoring.moveVelocitySelected := FALSE;
   cmSepaGripperAxisX.monitoring.stopSelected := FALSE;
   cmSepaGripperAxisX.monitoring.fastStopSelected := FALSE;
   cmSepaGripperAxisX.monitoring.torqueLimitingSelected := FALSE;
   cmSepaGripperAxisX.monitoring.homingSelected := FALSE;
   cmSepaGripperAxisX.monitoring.posRelativeSelected := FALSE;
   cmSepaGripperAxisX.monitoring.posAbsoluteSelected := FALSE;
   cmSepaGripperAxisX.monitoring.posSuperimposedSelected := FALSE;
   cmSepaGripperAxisX.monitoring.haltSuperimposedSelected := FALSE;
   cmSepaGripperAxisX.monitoring.commandBusy := FALSE;
   cmSepaGripperAxisX.monitoring.commandDone := FALSE;
   cmSepaGripperAxisX.monitoring.commandAborted := FALSE;
   cmSepaGripperAxisX.monitoring.homingCommandBusy := FALSE;
   cmSepaGripperAxisX.monitoring.homingCommandDone := FALSE;
   cmSepaGripperAxisX.monitoring.homingCommandAborted := FALSE;
   cmSepaGripperAxisX.monitoring.superimposedBusy := FALSE;
   cmSepaGripperAxisX.monitoring.superimposedDone := FALSE;
   cmSepaGripperAxisX.monitoring.superimposedAborted := FALSE;
   cmSepaGripperAxisX.monitoring.selectSetPosition := -1;
   cmSepaGripperAxisX.monitoring.selectionController := FALSE;
   cmSepaGripperAxisX.monitoring.interlockGeneral := TRUE;
   cmSepaGripperAxisX.monitoring.interlockJogForward := TRUE;
   cmSepaGripperAxisX.monitoring.interlockJogBackward := TRUE;
   cmSepaGripperAxisX.monitoring.interlockWarningGeneral := FALSE;
   cmSepaGripperAxisX.monitoring.interlockWarningJogForward := FALSE;
   cmSepaGripperAxisX.monitoring.interlockWarningJogBackward := FALSE;
   cmSepaGripperAxisX.monitoring.valid := TRUE;
   cmSepaGripperAxisX.monitoring.busy := TRUE;
   cmSepaGripperAxisX.monitoring.error := FALSE;
   cmSepaGripperAxisX.monitoring.status := 16#7002;
   cmSepaGripperAxisX.monitoring.subfunctionStatus := 16#0000;
   cmSepaGripperAxisX.monitoring.actualPosition := 100.0;
   cmSepaGripperAxisX.monitoring.actualSpeed := 0.0;
   cmSepaGripperAxisX.monitoring.speedUnit := 1062;
   cmSepaGripperAxisX.monitoring.positionUnit := 1013;
   cmSepaGripperAxisX.monitoring.axisStatus1 := 16#0200_10E1;
   cmSepaGripperAxisX.monitoring.axisStatus2 := 16#0000_0000;
   cmSepaGripperAxisX.monitoring.axisType := 1;
   cmSepaGripperAxisX.monitoring.maxVelocity := 2500.0;
   cmSepaGripperAxisX.monitoring.actualCurrent := 0.0;
   cmSepaGripperAxisX.monitoring.actualTorque := 0.0;
   cmSepaGripperAxisX.monitoring.velocityOverrideEnabled := FALSE;
   cmSepaGripperAxisX.monitoring.sinaParaError := FALSE;
   cmSepaGripperAxisX.monitoring.sinaParaStatus := 16#0000_0000;
   cmSepaGripperAxisX.configuration.referenceDesignator := WSTRING#'SepaGripperAxisX';
   cmSepaGripperAxisX.configuration.disableAlarms := FALSE;
   cmSepaGripperAxisX.configuration.masterControlPopUp := TRUE;
   cmSepaGripperAxisX.configuration.setPositions[0].position := 100.0;
   cmSepaGripperAxisX.configuration.setPositions[1].position := 400.0;
   cmSepaGripperAxisX.configuration.setPositions[2].position := 300.0;
   cmSepaGripperAxisX.configuration.setPositions[3].position := 150.0;
   cmSepaGripperAxisX.configuration.setPositions[4].position := 250.0;
   cmSepaGripperAxisX.configuration.setPositions[5].position := 100.0;
   cmSepaGripperAxisX.configuration.setPositions[6..15].position := 0.0;
   cmSepaGripperAxisX.configuration.setPositions[0..6].velocity := 100.0;
   cmSepaGripperAxisX.configuration.setPositions[7..15].velocity := -1.0;
   cmSepaGripperAxisX.configuration.setPositions[0..6].acceleration := 1000.0;
   cmSepaGripperAxisX.configuration.setPositions[7..15].acceleration := -1.0;
   cmSepaGripperAxisX.configuration.setPositions[0..6].deceleration := 1000.0;
   cmSepaGripperAxisX.configuration.setPositions[7..15].deceleration := -1.0;
   cmSepaGripperAxisX.configuration.setPositions[0..15]."name" := '';
   cmSepaGripperAxisZ.commandConfiguration.generalSettings.stopOnError := TRUE;
   cmSepaGripperAxisZ.commandConfiguration.generalSettings.resetWithRestart := FALSE;
   cmSepaGripperAxisZ.commandConfiguration.generalSettings.abortWaitingSyncCmd := TRUE;
   cmSepaGripperAxisZ.commandConfiguration.power.startMode := 1;
   cmSepaGripperAxisZ.commandConfiguration.power.stopMode := 0;
   cmSepaGripperAxisZ.commandConfiguration.power.syncMotionSimulation := FALSE;
   cmSepaGripperAxisZ.commandConfiguration.power.syncMotionSimulationExtendedMode := -1;
   cmSepaGripperAxisZ.commandConfiguration.jog.velocity := 20.0;
   cmSepaGripperAxisZ.commandConfiguration.jog.acceleration := -1.0;
   cmSepaGripperAxisZ.commandConfiguration.jog.deceleration := -1.0;
   cmSepaGripperAxisZ.commandConfiguration.jog.jerk := -1.0;
   cmSepaGripperAxisZ.commandConfiguration.jog.positionControlled := TRUE;
   cmSepaGripperAxisZ.commandConfiguration.jog.increment := 0.0;
   cmSepaGripperAxisZ.commandConfiguration.jog.mode := 0;
   cmSepaGripperAxisZ.commandConfiguration.moveVelocity.velocity := 0.0;
   cmSepaGripperAxisZ.commandConfiguration.moveVelocity.acceleration := -1.0;
   cmSepaGripperAxisZ.commandConfiguration.moveVelocity.deceleration := -1.0;
   cmSepaGripperAxisZ.commandConfiguration.moveVelocity.jerk := -1.0;
   cmSepaGripperAxisZ.commandConfiguration.moveVelocity.direction := 0;
   cmSepaGripperAxisZ.commandConfiguration.moveVelocity.positionControlled := TRUE;
   cmSepaGripperAxisZ.commandConfiguration.moveVelocity.velocityChangeOnTheFly := FALSE;
   cmSepaGripperAxisZ.commandConfiguration.stop.deceleration := -1.0;
   cmSepaGripperAxisZ.commandConfiguration.stop.jerk := -1.0;
   cmSepaGripperAxisZ.commandConfiguration.stop.abortAcceleration := FALSE;
   cmSepaGripperAxisZ.commandConfiguration.fastStop.deceleration := -1.0;
   cmSepaGripperAxisZ.commandConfiguration.fastStop.jerk := -1.0;
   cmSepaGripperAxisZ.commandConfiguration.fastStop.abortAcceleration := FALSE;
   cmSepaGripperAxisZ.commandConfiguration.fastStop.replaceStopPossible := FALSE;
   cmSepaGripperAxisZ.commandConfiguration.torqueLimiting.limit := -1.0;
   cmSepaGripperAxisZ.commandConfiguration.torqueLimiting.mode := 0;
   cmSepaGripperAxisZ.commandConfiguration.homing.position := 0.0;
   cmSepaGripperAxisZ.commandConfiguration.homing.mode := 0;
   cmSepaGripperAxisZ.commandConfiguration.homing.sensor := 0;
   cmSepaGripperAxisZ.commandConfiguration.homing.extendedMode := -1;
   cmSepaGripperAxisZ.commandConfiguration.homing.extendedModeTorqueLimit := 0.0;
   cmSepaGripperAxisZ.commandConfiguration.homing.extendedModeTargetPosition := 0.0;
   cmSepaGripperAxisZ.commandConfiguration.posRelative.distance := 0.0;
   cmSepaGripperAxisZ.commandConfiguration.posRelative.velocity := -1.0;
   cmSepaGripperAxisZ.commandConfiguration.posRelative.acceleration := -1.0;
   cmSepaGripperAxisZ.commandConfiguration.posRelative.deceleration := -1.0;
   cmSepaGripperAxisZ.commandConfiguration.posRelative.jerk := -1.0;
   cmSepaGripperAxisZ.commandConfiguration.posRelative.direction := 0;
   cmSepaGripperAxisZ.commandConfiguration.posAbsolute.position := 0.0;
   cmSepaGripperAxisZ.commandConfiguration.posAbsolute.velocity := -1.0;
   cmSepaGripperAxisZ.commandConfiguration.posAbsolute.acceleration := -1.0;
   cmSepaGripperAxisZ.commandConfiguration.posAbsolute.deceleration := -1.0;
   cmSepaGripperAxisZ.commandConfiguration.posAbsolute.jerk := -1.0;
   cmSepaGripperAxisZ.commandConfiguration.posAbsolute.direction := 1;
   cmSepaGripperAxisZ.commandConfiguration.posAbsolute.positionChangeOnTheFly := FALSE;
   cmSepaGripperAxisZ.commandConfiguration.posAbsolute.velocityChangeOnTheFly := FALSE;
   cmSepaGripperAxisZ.commandConfiguration.posSuperimposed.distance := 0.0;
   cmSepaGripperAxisZ.commandConfiguration.posSuperimposed.velocityDiff := -1.0;
   cmSepaGripperAxisZ.commandConfiguration.posSuperimposed.acceleration := -1.0;
   cmSepaGripperAxisZ.commandConfiguration.posSuperimposed.deceleration := -1.0;
   cmSepaGripperAxisZ.commandConfiguration.posSuperimposed.jerk := -1.0;
   cmSepaGripperAxisZ.commandConfiguration.posSuperimposed.direction := 0;
   cmSepaGripperAxisZ.commandConfiguration.haltSuperimposed.deceleration := -1.0;
